RoboDK station: kr30 cnc template half inch flat end mill - paulina 3.rdk

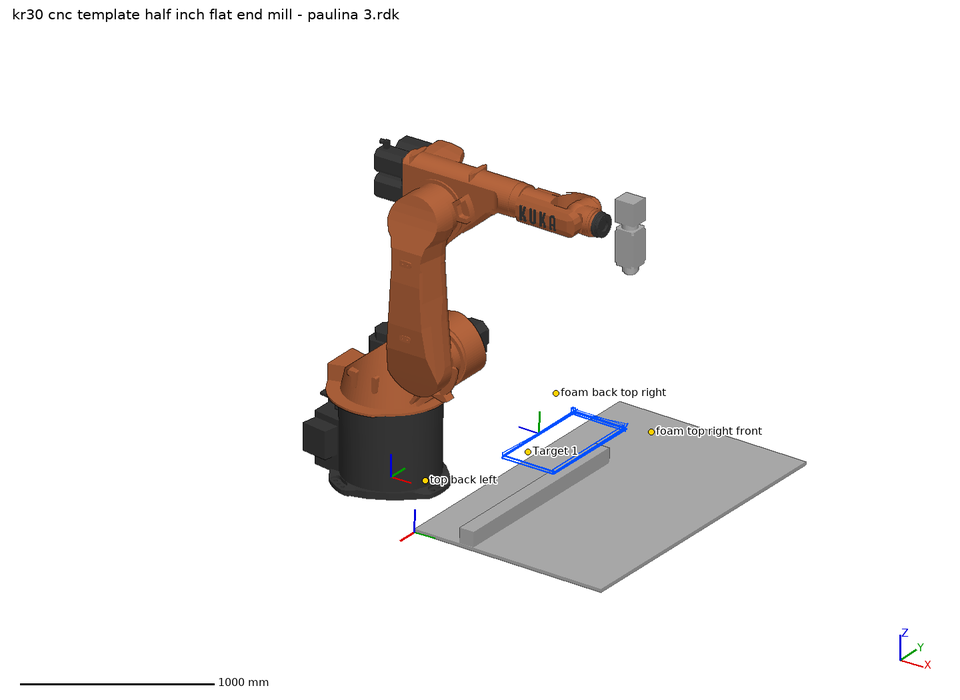
[picture v0: the station drawn from its stored meshes, robots at their saved joint values, targets as dots, program paths as lines]
Station kr30 cnc template half inch flat end mill - paulina 3. Poses are relative to the parent item; angles as X-Y-Z fixed-axis rotations.
  - frame KUKA KR 30 HA Base at (0, 0, 0) mm
    - robot KUKA KR 30 HA: 6 axes, payload 30 kg, reach 2033 mm, repeatability 0.05 mm, weight 665 kg
        modified DH rows (alpha deg, a mm, theta deg, d mm): 0, 0, 0, 815; -90, 350, 0, 0; 0, 850, -90, 0; -90, 145, 0, 820; 90, 0, 0, 0; -90, 0, 180, 170
        joint limits [-185, -135, -120, -350, -119, -350] to [185, 35, 158, 350, 119, 350]; home [0, -90, 90, 0, 0, 0]; saved at [0, -90, 90, 0, 0, 0]
      - tool rc90 spindle mm, TCP at (337.31, -2.2, 160.57) mm, size 110 x 421.3 x 118 mm, geometry from rc90 spindle mm.stl
    - frame Tabletop at (921.82, -1104.91, 385) mm, rotated rx -0.93 ry -0.21 rz -89.9 deg
      - object tabletop CHECK HEIGHT at (-1839.9, 0, 0) mm, size 1839.9 x 1168.4 x 19 mm, geometry from kr30 tabletop mm.stl
      - object kr30 pipe jig base at (-1220, -610.6, 0) mm, size 1217.6 x 88.9 x 88.9 mm, geometry from kr30 pipe jig base.stl
      - frame Frame 3 at (-550, 390, 460) mm, rotated rx 90 ry 0 rz 0 deg
        - target Target 1 (Cartesian target) at (324.46, 69.12, -153.95) mm, rotated rx -179.9 ry 0.14 rz -89.96 deg; joints [37.245, -66.694, 101.534, 53.768, -48.608, -41.204] of KUKA KR 30 HA
    - target foam back top right (Cartesian target) at (1197.65, -230.62, 906.79) mm, rotated rx -15.53 ry 90 rz -15.53 deg; joints [14.757, -102.447, 141.256, 22.791, -41.102, -17.568] of KUKA KR 30 HA
    - target foam top right front (Cartesian target) at (1797.45, -230.62, 850.68) mm, rotated rx -15.58 ry 90 rz -15.58 deg; joints [8.85, -62.405, 99.608, 14.434, -38.093, -11.451] of KUKA KR 30 HA
    - target top back left (Cartesian target) at (1223.08, -1440.01, 894.96) mm, rotated rx 58.97 ry 90 rz 58.97 deg; joints [58.171, -50.232, 76.73, 74.515, -61.834, -59.599] of KUKA KR 30 HA
  - machining project Machining Settings: C:/Users/Research Office/Downloads/b4.apt | rotZ(0) | rotX(0)*rotY(0) | roty(-90) | onStart | onPathStart | onApproach | onPoint | onRetract | onFinish | SetTool(%1) | onPathFinish
  - program Machining (938 instructions, listed below)
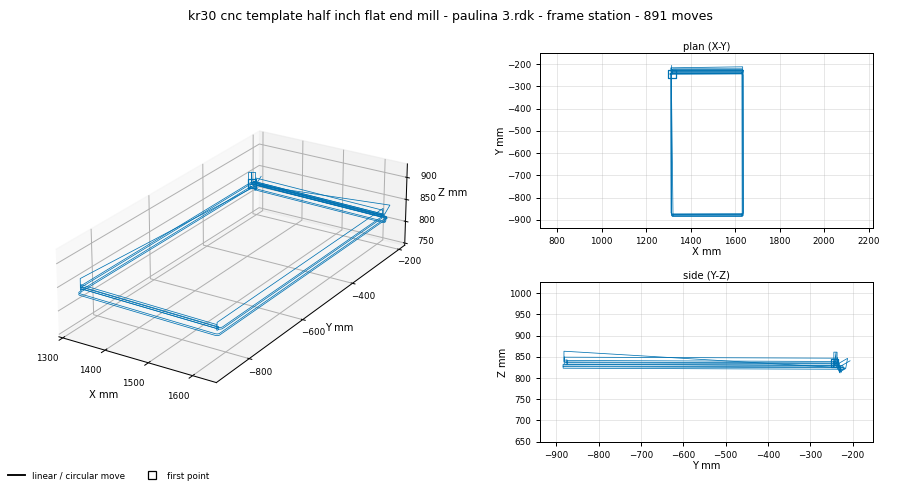
[picture p0: tool path of kr30 cnc template half inch flat end mill - paulina 3.rdk in frame station, 891 of 891 moves have a stored position in this frame; points joined in program order, loops and branches not executed]

--- program Machining (robot KUKA KR 30 HA) ---
  Smooth(10)
  Print: /'1001'
  Print: /''
  Print: /'Contour3'
  Call SetTool(1)
  Set speed (200.0 mm/s)
  Set Ref.: Frame 3
  Set Tool: rc90 spindle mm
  Show rc90 spindle mm
  MoveJ 1 to (-309.78, 0.83, 2.88) mm, rotated rx -179.88 ry 0.12 rz -89.97 deg; joints [13.585, -90.541, 136.338, 18.844, -46.545, -12.771]
  MoveL 2 to (-313.47, 25.53, 7.11) mm, rotated rx -179.9 ry 0 rz -90 deg; joints [13.435, -92.009, 135.635, -160.591, 44.341, 166.292]
  MoveL 3 to (-313.47, 25.53, 7.11) mm, rotated rx -179.9 ry 0 rz -90 deg; joints [13.435, -92.009, 135.635, -160.591, 44.341, 166.292]
  Set speed (200.0 mm/s)
  MoveL 4 to (-313.47, 10.99, 7.11) mm, rotated rx -179.9 ry 0 rz -90 deg; joints [13.441, -91.344, 136.203, -160.99, 45.507, 166.861]
  Set speed (50.0 mm/s)
  MoveL 5 to (-313.47, 4.79, 7.11) mm, rotated rx -179.9 ry 0 rz -90 deg; joints [13.444, -91.052, 136.44, -161.153, 46.008, 167.098]
  MoveL 6 to (-312.33, 3.53, 6.55) mm, rotated rx -179.9 ry 0 rz -90 deg; joints [13.5, -90.937, 136.434, -161.112, 46.125, 167.095]
  Set speed (100.0 mm/s)
  MoveL 7 to (-308.58, 3.52, 4.75) mm, rotated rx -179.9 ry 0 rz -90 deg; joints [13.681, -90.756, 136.258, -160.868, 46.171, 166.931]
  MoveC 8 to (-307.9, 3.53, 3.89) mm, rotated rx -179.9 ry 0 rz -90 deg; joints [13.707, -90.688, 136.192, -160.834, 46.179, 166.908] to (-308.14, 3.52, 2.82) mm, rotated rx -179.9 ry 0 rz -90 deg; joints [13.68, -90.62, 136.127, -160.872, 46.175, 166.934]
  MoveL 9 to (-308.14, 3.52, 2.82) mm, rotated rx -179.9 ry 0 rz -90 deg; joints [13.68, -90.62, 136.127, -160.872, 46.175, 166.934]
  MoveL 10 to (-308.36, 3.52, 2.5) mm, rotated rx -179.9 ry 0 rz -90 deg; joints [13.663, -90.603, 136.11, -160.894, 46.171, 166.95]
  MoveL 11 to (-308.56, 3.53, 2.18) mm, rotated rx -179.9 ry 0 rz -90 deg; joints [13.648, -90.584, 136.093, -160.915, 46.169, 166.964]
  MoveL 12 to (-308.73, 3.52, 1.86) mm, rotated rx -179.9 ry 0 rz -90 deg; joints [13.635, -90.566, 136.075, -160.934, 46.166, 166.977]
  MoveL 13 to (-308.88, 3.53, 1.54) mm, rotated rx -179.9 ry 0 rz -90 deg; joints [13.622, -90.547, 136.057, -160.951, 46.164, 166.989]
  MoveL 14 to (-309.02, 3.52, 1.19) mm, rotated rx -179.9 ry 0 rz -90 deg; joints [13.61, -90.526, 136.036, -160.967, 46.162, 167]
  MoveL 15 to (-309.14, 3.53, 0.84) mm, rotated rx -179.9 ry 0 rz -90 deg; joints [13.599, -90.505, 136.016, -160.983, 46.16, 167.011]
  MoveL 16 to (-309.23, 3.53, 0.5) mm, rotated rx -179.9 ry 0 rz -90 deg; joints [13.589, -90.483, 135.995, -160.996, 46.159, 167.02]
  MoveL 17 to (-309.31, 3.53, 0.15) mm, rotated rx -179.9 ry 0 rz -90 deg; joints [13.58, -90.461, 135.973, -161.008, 46.157, 167.029]
  MoveL 18 to (-309.36, 3.53, -0.2) mm, rotated rx -179.9 ry 0 rz -90 deg; joints [13.573, -90.438, 135.952, -161.018, 46.156, 167.036]
  MoveL 19 to (-309.4, 3.52, -0.55) mm, rotated rx -179.9 ry 0 rz -90 deg; joints [13.566, -90.416, 135.93, -161.027, 46.156, 167.042]
  MoveL 20 to (-309.41, 3.53, -1.25) mm, rotated rx -179.9 ry 0 rz -90 deg; joints [13.556, -90.369, 135.885, -161.041, 46.155, 167.052]
  MoveL 21 to (-309.41, 3.52, -310.99) mm, rotated rx -179.9 ry 0 rz -90 deg; joints [10.396, -71.401, 113.657, -164.475, 42.367, 168.785]
  MoveL 22 to (-309.4, 3.52, -311.68) mm, rotated rx -179.9 ry 0 rz -90 deg; joints [10.391, -71.36, 113.601, -164.478, 42.352, 168.784]
  MoveL 23 to (-309.36, 3.52, -312.03) mm, rotated rx -179.9 ry 0 rz -90 deg; joints [10.39, -71.34, 113.573, -164.478, 42.344, 168.783]
  MoveL 24 to (-309.31, 3.52, -312.38) mm, rotated rx -179.9 ry 0 rz -90 deg; joints [10.389, -71.319, 113.545, -164.476, 42.337, 168.78]
  MoveL 25 to (-309.23, 3.53, -312.73) mm, rotated rx -179.9 ry 0 rz -90 deg; joints [10.39, -71.298, 113.516, -164.473, 42.329, 168.777]
  MoveL 26 to (-309.14, 3.52, -313.08) mm, rotated rx -179.9 ry 0 rz -90 deg; joints [10.391, -71.276, 113.487, -164.469, 42.322, 168.772]
  MoveL 27 to (-309.02, 3.52, -313.43) mm, rotated rx -179.9 ry 0 rz -90 deg; joints [10.393, -71.255, 113.457, -164.464, 42.315, 168.767]
  MoveL 28 to (-308.88, 3.52, -313.78) mm, rotated rx -179.9 ry 0 rz -90 deg; joints [10.396, -71.233, 113.427, -164.457, 42.308, 168.76]
  MoveL 29 to (-308.73, 3.53, -314.1) mm, rotated rx -179.9 ry 0 rz -90 deg; joints [10.4, -71.213, 113.4, -164.449, 42.301, 168.753]
  MoveL 30 to (-308.56, 3.52, -314.42) mm, rotated rx -179.9 ry 0 rz -90 deg; joints [10.405, -71.192, 113.372, -164.439, 42.295, 168.745]
  MoveL 31 to (-308.36, 3.52, -314.73) mm, rotated rx -179.9 ry 0 rz -90 deg; joints [10.411, -71.172, 113.343, -164.429, 42.289, 168.736]
  MoveL 32 to (-308.14, 3.52, -315.05) mm, rotated rx -179.9 ry 0 rz -90 deg; joints [10.418, -71.151, 113.315, -164.416, 42.283, 168.725]
  MoveL 33 to (-307.96, 3.52, -315.28) mm, rotated rx -179.9 ry 0 rz -90 deg; joints [10.424, -71.136, 113.294, -164.406, 42.278, 168.717]
  MoveL 34 to (-307.77, 3.53, -315.5) mm, rotated rx -179.9 ry 0 rz -90 deg; joints [10.43, -71.121, 113.274, -164.395, 42.274, 168.708]
  MoveL 35 to (-307.55, 3.53, -315.73) mm, rotated rx -179.9 ry 0 rz -90 deg; joints [10.438, -71.105, 113.252, -164.382, 42.27, 168.697]
  MoveL 36 to (-307.32, 3.53, -315.94) mm, rotated rx -179.9 ry 0 rz -90 deg; joints [10.445, -71.09, 113.232, -164.369, 42.266, 168.687]
  MoveL 37 to (-306.92, 3.52, -316.28) mm, rotated rx -179.9 ry 0 rz -90 deg; joints [10.46, -71.066, 113.198, -164.346, 42.26, 168.668]
  MoveL 38 to (-306.51, 3.53, -316.57) mm, rotated rx -179.9 ry 0 rz -90 deg; joints [10.475, -71.045, 113.17, -164.321, 42.256, 168.649]
  MoveL 39 to (-306.22, 3.52, -316.74) mm, rotated rx -179.9 ry 0 rz -90 deg; joints [10.486, -71.032, 113.151, -164.304, 42.253, 168.635]
  MoveL 40 to (-305.93, 3.52, -316.9) mm, rotated rx -179.9 ry 0 rz -90 deg; joints [10.497, -71.02, 113.134, -164.287, 42.251, 168.621]
  MoveL 41 to (-305.64, 3.52, -317.04) mm, rotated rx -179.9 ry 0 rz -90 deg; joints [10.508, -71.009, 113.119, -164.269, 42.249, 168.608]
  MoveL 42 to (-305.35, 3.52, -317.16) mm, rotated rx -179.9 ry 0 rz -90 deg; joints [10.519, -70.999, 113.105, -164.251, 42.248, 168.594]
  MoveL 43 to (-305, 3.52, -317.28) mm, rotated rx -179.9 ry 0 rz -90 deg; joints [10.533, -70.988, 113.09, -164.23, 42.246, 168.578]
  MoveL 44 to (-304.65, 3.52, -317.38) mm, rotated rx -179.9 ry 0 rz -90 deg; joints [10.547, -70.978, 113.076, -164.209, 42.245, 168.562]
  MoveL 45 to (-304.3, 3.52, -317.46) mm, rotated rx -179.9 ry 0 rz -90 deg; joints [10.561, -70.97, 113.065, -164.187, 42.245, 168.545]
  MoveL 46 to (-303.95, 3.53, -317.52) mm, rotated rx -179.9 ry 0 rz -90 deg; joints [10.575, -70.963, 113.055, -164.166, 42.245, 168.529]
  MoveL 47 to (-303.6, 3.52, -317.56) mm, rotated rx -179.9 ry 0 rz -90 deg; joints [10.59, -70.956, 113.046, -164.144, 42.246, 168.513]
  MoveL 48 to (-303.26, 3.52, -317.58) mm, rotated rx -179.9 ry 0 rz -90 deg; joints [10.604, -70.952, 113.039, -164.122, 42.247, 168.496]
  MoveL 49 to (-302.56, 3.53, -317.59) mm, rotated rx -179.9 ry 0 rz -90 deg; joints [10.634, -70.944, 113.028, -164.078, 42.25, 168.464]
  MoveL 50 to (315.11, 3.52, -317.59) mm, rotated rx -179.9 ry 0 rz -90 deg; joints [33.369, -56.917, 91.684, -130.086, 45.952, 141.267]
  MoveL 51 to (315.8, 3.53, -317.58) mm, rotated rx -179.9 ry 0 rz -90 deg; joints [33.39, -56.894, 91.646, -130.052, 45.956, 141.236]
  MoveL 52 to (316.15, 3.53, -317.56) mm, rotated rx -179.9 ry 0 rz -90 deg; joints [33.401, -56.883, 91.628, -130.035, 45.958, 141.221]
  MoveL 53 to (316.5, 3.52, -317.52) mm, rotated rx -179.9 ry 0 rz -90 deg; joints [33.413, -56.873, 91.612, -130.018, 45.961, 141.206]
  MoveL 54 to (316.82, 3.52, -317.46) mm, rotated rx -179.9 ry 0 rz -90 deg; joints [33.423, -56.865, 91.599, -130.003, 45.965, 141.192]
  MoveL 55 to (317.13, 3.52, -317.39) mm, rotated rx -179.9 ry 0 rz -90 deg; joints [33.434, -56.858, 91.588, -129.988, 45.969, 141.18]
  MoveL 56 to (317.45, 3.53, -317.3) mm, rotated rx -179.9 ry 0 rz -90 deg; joints [33.446, -56.852, 91.578, -129.973, 45.974, 141.167]
  MoveL 57 to (317.76, 3.52, -317.2) mm, rotated rx -179.9 ry 0 rz -90 deg; joints [33.457, -56.847, 91.569, -129.957, 45.979, 141.155]
  MoveL 58 to (318.08, 3.52, -317.07) mm, rotated rx -179.9 ry 0 rz -90 deg; joints [33.469, -56.843, 91.562, -129.942, 45.985, 141.143]
  MoveL 59 to (318.4, 3.52, -316.93) mm, rotated rx -179.9 ry 0 rz -90 deg; joints [33.482, -56.839, 91.557, -129.927, 45.991, 141.131]
  MoveL 60 to (318.71, 3.52, -316.76) mm, rotated rx -179.9 ry 0 rz -90 deg; joints [33.495, -56.837, 91.553, -129.912, 45.998, 141.12]
  MoveL 61 to (319.03, 3.53, -316.57) mm, rotated rx -179.9 ry 0 rz -90 deg; joints [33.508, -56.836, 91.551, -129.897, 46.006, 141.109]
  MoveL 62 to (319.29, 3.52, -316.39) mm, rotated rx -179.9 ry 0 rz -90 deg; joints [33.52, -56.837, 91.552, -129.884, 46.013, 141.101]
  MoveL 63 to (319.63, 3.52, -316.13) mm, rotated rx -179.9 ry 0 rz -90 deg; joints [33.535, -56.839, 91.554, -129.868, 46.024, 141.09]
  MoveL 64 to (319.96, 3.52, -315.83) mm, rotated rx -179.9 ry 0 rz -90 deg; joints [33.552, -56.843, 91.56, -129.852, 46.035, 141.081]
  MoveL 65 to (320.32, 3.53, -315.46) mm, rotated rx -179.9 ry 0 rz -90 deg; joints [33.57, -56.85, 91.571, -129.835, 46.049, 141.071]
  MoveL 66 to (320.63, 3.52, -315.08) mm, rotated rx -179.9 ry 0 rz -90 deg; joints [33.587, -56.859, 91.585, -129.82, 46.063, 141.064]
  MoveL 67 to (320.86, 3.52, -314.76) mm, rotated rx -179.9 ry 0 rz -90 deg; joints [33.601, -56.868, 91.599, -129.809, 46.075, 141.059]
  MoveL 68 to (321.07, 3.52, -314.43) mm, rotated rx -179.9 ry 0 rz -90 deg; joints [33.614, -56.878, 91.615, -129.8, 46.087, 141.056]
  MoveL 69 to (321.24, 3.53, -314.1) mm, rotated rx -179.9 ry 0 rz -90 deg; joints [33.626, -56.889, 91.632, -129.792, 46.098, 141.054]
  MoveL 70 to (321.4, 3.52, -313.78) mm, rotated rx -179.9 ry 0 rz -90 deg; joints [33.637, -56.9, 91.65, -129.784, 46.11, 141.053]
  MoveL 71 to (321.54, 3.52, -313.43) mm, rotated rx -179.9 ry 0 rz -90 deg; joints [33.648, -56.914, 91.671, -129.778, 46.122, 141.053]
  MoveL 72 to (321.66, 3.52, -313.08) mm, rotated rx -179.9 ry 0 rz -90 deg; joints [33.659, -56.928, 91.694, -129.773, 46.134, 141.054]
  MoveL 73 to (321.75, 3.52, -312.73) mm, rotated rx -179.9 ry 0 rz -90 deg; joints [33.669, -56.943, 91.717, -129.768, 46.145, 141.056]
  MoveL 74 to (321.83, 3.52, -312.38) mm, rotated rx -179.9 ry 0 rz -90 deg; joints [33.678, -56.958, 91.742, -129.765, 46.157, 141.059]
  MoveL 75 to (321.88, 3.52, -312.03) mm, rotated rx -179.9 ry 0 rz -90 deg; joints [33.687, -56.974, 91.767, -129.763, 46.169, 141.062]
  MoveL 76 to (321.91, 3.52, -311.68) mm, rotated rx -179.9 ry 0 rz -90 deg; joints [33.695, -56.991, 91.794, -129.761, 46.18, 141.067]
  MoveL 77 to (321.93, 3.53, -310.99) mm, rotated rx -179.9 ry 0 rz -90 deg; joints [33.71, -57.027, 91.851, -129.761, 46.203, 141.079]
  MoveL 78 to (321.93, 3.52, -1.25) mm, rotated rx -179.9 ry 0 rz -90 deg; joints [41.195, -71.851, 113.68, -126.635, 55.146, 143.485]
  MoveL 79 to (321.91, 3.52, -0.55) mm, rotated rx -179.9 ry 0 rz -90 deg; joints [41.215, -71.883, 113.723, -126.623, 55.164, 143.485]
  MoveL 80 to (321.88, 3.52, -0.2) mm, rotated rx -179.9 ry 0 rz -90 deg; joints [41.224, -71.9, 113.746, -126.617, 55.173, 143.486]
  MoveL 81 to (321.83, 3.52, 0.15) mm, rotated rx -179.9 ry 0 rz -90 deg; joints [41.232, -71.918, 113.77, -126.613, 55.181, 143.488]
  MoveL 82 to (321.75, 3.52, 0.5) mm, rotated rx -179.9 ry 0 rz -90 deg; joints [41.239, -71.936, 113.795, -126.609, 55.19, 143.49]
  MoveL 83 to (321.66, 3.53, 0.84) mm, rotated rx -179.9 ry 0 rz -90 deg; joints [41.246, -71.956, 113.821, -126.606, 55.198, 143.493]
  MoveL 84 to (321.54, 3.53, 1.19) mm, rotated rx -179.9 ry 0 rz -90 deg; joints [41.252, -71.976, 113.848, -126.604, 55.206, 143.496]
  MoveL 85 to (321.4, 3.53, 1.54) mm, rotated rx -179.9 ry 0 rz -90 deg; joints [41.258, -71.997, 113.877, -126.603, 55.213, 143.501]
  MoveL 86 to (321.24, 3.52, 1.87) mm, rotated rx -179.9 ry 0 rz -90 deg; joints [41.262, -72.017, 113.904, -126.602, 55.22, 143.505]
  MoveL 87 to (321.07, 3.52, 2.19) mm, rotated rx -179.9 ry 0 rz -90 deg; joints [41.266, -72.039, 113.934, -126.603, 55.227, 143.511]
  MoveL 88 to (320.86, 3.52, 2.52) mm, rotated rx -179.9 ry 0 rz -90 deg; joints [41.269, -72.061, 113.964, -126.605, 55.233, 143.517]
  MoveL 89 to (320.63, 3.52, 2.85) mm, rotated rx -179.9 ry 0 rz -90 deg; joints [41.27, -72.085, 113.996, -126.608, 55.239, 143.524]
  MoveL 90 to (320.32, 3.52, 3.22) mm, rotated rx -179.9 ry 0 rz -90 deg; joints [41.271, -72.114, 114.035, -126.613, 55.246, 143.534]
  MoveL 91 to (319.96, 3.52, 3.6) mm, rotated rx -179.9 ry 0 rz -90 deg; joints [41.27, -72.145, 114.077, -126.62, 55.252, 143.545]
  MoveL 92 to (319.63, 3.53, 3.89) mm, rotated rx -179.9 ry 0 rz -90 deg; joints [41.268, -72.171, 114.113, -126.628, 55.256, 143.556]
  MoveL 93 to (319.29, 3.52, 4.15) mm, rotated rx -179.9 ry 0 rz -90 deg; joints [41.264, -72.196, 114.146, -126.636, 55.259, 143.566]
  MoveL 94 to (319.03, 3.53, 4.33) mm, rotated rx -179.9 ry 0 rz -90 deg; joints [41.261, -72.214, 114.171, -126.643, 55.261, 143.575]
  MoveL 95 to (318.71, 3.52, 4.52) mm, rotated rx -179.9 ry 0 rz -90 deg; joints [41.256, -72.235, 114.2, -126.652, 55.263, 143.585]
  MoveL 96 to (318.4, 3.52, 4.69) mm, rotated rx -179.9 ry 0 rz -90 deg; joints [41.25, -72.255, 114.226, -126.661, 55.264, 143.594]
  MoveL 97 to (318.08, 3.53, 4.84) mm, rotated rx -179.9 ry 0 rz -90 deg; joints [41.244, -72.274, 114.252, -126.671, 55.264, 143.604]
  MoveL 98 to (317.76, 3.53, 4.96) mm, rotated rx -179.9 ry 0 rz -90 deg; joints [41.237, -72.291, 114.276, -126.681, 55.264, 143.614]
  MoveL 99 to (317.45, 3.52, 5.07) mm, rotated rx -179.9 ry 0 rz -90 deg; joints [41.23, -72.308, 114.3, -126.692, 55.263, 143.624]
  MoveL 100 to (317.13, 3.53, 5.16) mm, rotated rx -179.9 ry 0 rz -90 deg; joints [41.222, -72.325, 114.322, -126.703, 55.262, 143.634]
  MoveL 101 to (316.82, 3.52, 5.23) mm, rotated rx -179.9 ry 0 rz -90 deg; joints [41.214, -72.34, 114.343, -126.714, 55.261, 143.644]
  MoveL 102 to (316.5, 3.52, 5.28) mm, rotated rx -179.9 ry 0 rz -90 deg; joints [41.205, -72.355, 114.363, -126.725, 55.259, 143.654]
  MoveL 103 to (316.15, 3.53, 5.32) mm, rotated rx -179.9 ry 0 rz -90 deg; joints [41.195, -72.37, 114.384, -126.739, 55.256, 143.665]
  MoveL 104 to (315.8, 3.53, 5.35) mm, rotated rx -179.9 ry 0 rz -90 deg; joints [41.184, -72.385, 114.404, -126.752, 55.253, 143.676]
  MoveL 105 to (315.11, 3.53, 5.35) mm, rotated rx -179.9 ry 0 rz -90 deg; joints [41.162, -72.412, 114.441, -126.78, 55.245, 143.699]
  MoveL 106 to (-302.56, 3.53, 5.35) mm, rotated rx -179.9 ry 0 rz -90 deg; joints [14.019, -90.699, 136.199, -160.413, 46.247, 166.621]
  MoveL 107 to (-303.26, 3.53, 5.35) mm, rotated rx -179.9 ry 0 rz -90 deg; joints [13.981, -90.71, 136.21, -160.465, 46.238, 166.656]
  MoveL 108 to (-303.6, 3.52, 5.33) mm, rotated rx -179.9 ry 0 rz -90 deg; joints [13.961, -90.714, 136.215, -160.491, 46.234, 166.674]
  MoveL 109 to (-303.95, 3.52, 5.29) mm, rotated rx -179.9 ry 0 rz -90 deg; joints [13.942, -90.717, 136.218, -160.517, 46.229, 166.692]
  MoveL 110 to (-304.3, 3.53, 5.23) mm, rotated rx -179.9 ry 0 rz -90 deg; joints [13.922, -90.719, 136.22, -160.544, 46.225, 166.71]
  MoveL 111 to (-304.65, 3.53, 5.15) mm, rotated rx -179.9 ry 0 rz -90 deg; joints [13.902, -90.72, 136.221, -160.571, 46.22, 166.728]
  MoveL 112 to (-305, 3.53, 5.05) mm, rotated rx -179.9 ry 0 rz -90 deg; joints [13.881, -90.718, 136.22, -160.599, 46.216, 166.747]
  MoveL 113 to (-305.35, 3.52, 4.92) mm, rotated rx -179.9 ry 0 rz -90 deg; joints [13.861, -90.716, 136.217, -160.627, 46.211, 166.766]
  MoveL 114 to (-305.64, 3.53, 4.8) mm, rotated rx -179.9 ry 0 rz -90 deg; joints [13.843, -90.713, 136.214, -160.65, 46.208, 166.783]
  MoveL 115 to (-305.93, 3.53, 4.67) mm, rotated rx -179.9 ry 0 rz -90 deg; joints [13.825, -90.708, 136.21, -160.674, 46.204, 166.799]
  MoveL 116 to (-306.22, 3.52, 4.51) mm, rotated rx -179.9 ry 0 rz -90 deg; joints [13.807, -90.702, 136.205, -160.699, 46.2, 166.816]
  MoveL 117 to (-306.51, 3.52, 4.33) mm, rotated rx -179.9 ry 0 rz -90 deg; joints [13.789, -90.695, 136.198, -160.723, 46.196, 166.833]
  MoveL 118 to (-306.92, 3.53, 4.05) mm, rotated rx -179.9 ry 0 rz -90 deg; joints [13.763, -90.683, 136.186, -160.759, 46.191, 166.857]
  MoveL 119 to (-307.32, 3.53, 3.71) mm, rotated rx -179.9 ry 0 rz -90 deg; joints [13.736, -90.667, 136.171, -160.795, 46.186, 166.882]
  MoveL 120 to (-307.55, 3.52, 3.5) mm, rotated rx -179.9 ry 0 rz -90 deg; joints [13.721, -90.656, 136.161, -160.816, 46.183, 166.896]
  MoveL 121 to (-307.77, 3.52, 3.26) mm, rotated rx -179.9 ry 0 rz -90 deg; joints [13.706, -90.644, 136.15, -160.836, 46.18, 166.91]
  MoveL 122 to (-307.96, 3.53, 3.04) mm, rotated rx -179.9 ry 0 rz -90 deg; joints [13.692, -90.632, 136.138, -160.855, 46.177, 166.923]
  MoveL 123 to (-308.14, 3.52, 2.82) mm, rotated rx -179.9 ry 0 rz -90 deg; joints [13.68, -90.62, 136.127, -160.872, 46.175, 166.934]
  MoveC 124 to (-309.89, 3.53, 2.59) mm, rotated rx -179.9 ry 0 rz -90 deg; joints [13.581, -90.633, 136.14, -161.006, 46.153, 167.026] to (-310.17, 3.53, 4.33) mm, rotated rx -179.9 ry 0 rz -90 deg; joints [13.589, -90.754, 136.257, -160.994, 46.15, 167.017]
  MoveL 125 to (-310.17, 3.52, 4.33) mm, rotated rx -179.9 ry 0 rz -90 deg; joints [13.589, -90.754, 136.257, -160.994, 46.15, 167.017]
  MoveL 126 to (-309.48, 3.53, 5.32) mm, rotated rx -179.9 ry 0 rz -90 deg; joints [13.64, -90.809, 136.31, -160.924, 46.16, 166.968]
  Set speed (50.0 mm/s)
  MoveL 127 to (-309.48, 1.27, 5.32) mm, rotated rx -179.9 ry 0 rz -90 deg; joints [13.641, -90.701, 136.395, -160.983, 46.342, 167.055]
  MoveL 128 to (-308.44, 0, 4.59) mm, rotated rx -179.9 ry 0 rz -90 deg; joints [13.688, -90.575, 136.379, -160.953, 46.457, 167.061]
  Set speed (100.0 mm/s)
  MoveC 129 to (-307.92, 0, 3.77) mm, rotated rx -179.9 ry 0 rz -90 deg; joints [13.706, -90.512, 136.317, -160.93, 46.462, 167.046] to (-308.14, 0, 2.82) mm, rotated rx -179.9 ry 0 rz -90 deg; joints [13.681, -90.452, 136.259, -160.964, 46.459, 167.069]
  MoveL 130 to (-308.14, 0, 2.82) mm, rotated rx -179.9 ry 0 rz -90 deg; joints [13.681, -90.452, 136.259, -160.964, 46.459, 167.069]
  MoveL 131 to (-308.36, 0, 2.5) mm, rotated rx -179.9 ry 0 rz -90 deg; joints [13.665, -90.435, 136.242, -160.986, 46.456, 167.084]
  MoveL 132 to (-308.56, 0, 2.18) mm, rotated rx -179.9 ry 0 rz -90 deg; joints [13.65, -90.417, 136.225, -161.007, 46.453, 167.098]
  MoveL 133 to (-308.73, 0, 1.86) mm, rotated rx -179.9 ry 0 rz -90 deg; joints [13.636, -90.398, 136.207, -161.025, 46.45, 167.111]
  MoveL 134 to (-308.88, 0, 1.54) mm, rotated rx -179.9 ry 0 rz -90 deg; joints [13.624, -90.379, 136.189, -161.042, 46.448, 167.123]
  MoveL 135 to (-309.02, 0, 1.19) mm, rotated rx -179.9 ry 0 rz -90 deg; joints [13.611, -90.358, 136.169, -161.059, 46.446, 167.134]
  MoveL 136 to (-309.14, 0, 0.84) mm, rotated rx -179.9 ry 0 rz -90 deg; joints [13.6, -90.337, 136.148, -161.074, 46.444, 167.144]
  MoveL 137 to (-309.23, 0, 0.5) mm, rotated rx -179.9 ry 0 rz -90 deg; joints [13.591, -90.315, 136.127, -161.087, 46.443, 167.154]
  MoveL 138 to (-309.31, 0, 0.15) mm, rotated rx -179.9 ry 0 rz -90 deg; joints [13.582, -90.293, 136.106, -161.099, 46.441, 167.162]
  MoveL 139 to (-309.36, 0, -0.2) mm, rotated rx -179.9 ry 0 rz -90 deg; joints [13.574, -90.271, 136.084, -161.109, 46.44, 167.169]
  MoveL 140 to (-309.4, 0, -0.55) mm, rotated rx -179.9 ry 0 rz -90 deg; joints [13.568, -90.248, 136.062, -161.118, 46.439, 167.175]
  MoveL 141 to (-309.41, 0, -1.25) mm, rotated rx -179.9 ry 0 rz -90 deg; joints [13.558, -90.202, 136.017, -161.132, 46.438, 167.185]
  MoveL 142 to (-309.41, 0, -310.99) mm, rotated rx -179.9 ry 0 rz -90 deg; joints [10.397, -71.274, 113.767, -164.543, 42.596, 168.878]
  MoveL 143 to (-309.4, 0, -311.68) mm, rotated rx -179.9 ry 0 rz -90 deg; joints [10.392, -71.233, 113.711, -164.546, 42.581, 168.877]
  MoveL 144 to (-309.36, 0, -312.03) mm, rotated rx -179.9 ry 0 rz -90 deg; joints [10.391, -71.212, 113.683, -164.546, 42.573, 168.876]
  MoveL 145 to (-309.31, 0, -312.38) mm, rotated rx -179.9 ry 0 rz -90 deg; joints [10.39, -71.191, 113.655, -164.544, 42.566, 168.873]
  MoveL 146 to (-309.23, 0, -312.73) mm, rotated rx -179.9 ry 0 rz -90 deg; joints [10.391, -71.17, 113.626, -164.541, 42.558, 168.869]
  MoveL 147 to (-309.14, 0, -313.08) mm, rotated rx -179.9 ry 0 rz -90 deg; joints [10.392, -71.149, 113.597, -164.537, 42.551, 168.865]
  MoveL 148 to (-309.02, 0, -313.43) mm, rotated rx -179.9 ry 0 rz -90 deg; joints [10.394, -71.127, 113.567, -164.531, 42.544, 168.86]
  MoveL 149 to (-308.88, 0, -313.78) mm, rotated rx -179.9 ry 0 rz -90 deg; joints [10.397, -71.106, 113.537, -164.524, 42.537, 168.853]
  MoveL 150 to (-308.73, 0, -314.1) mm, rotated rx -179.9 ry 0 rz -90 deg; joints [10.401, -71.086, 113.51, -164.517, 42.53, 168.846]
  MoveL 151 to (-308.56, 0, -314.42) mm, rotated rx -179.9 ry 0 rz -90 deg; joints [10.406, -71.065, 113.482, -164.508, 42.524, 168.838]
  MoveL 152 to (-308.36, 0, -314.73) mm, rotated rx -179.9 ry 0 rz -90 deg; joints [10.412, -71.045, 113.453, -164.497, 42.517, 168.829]
  MoveL 153 to (-308.14, 0, -315.05) mm, rotated rx -179.9 ry 0 rz -90 deg; joints [10.419, -71.024, 113.425, -164.484, 42.511, 168.818]
  MoveL 154 to (-307.96, 0, -315.28) mm, rotated rx -179.9 ry 0 rz -90 deg; joints [10.425, -71.009, 113.404, -164.474, 42.507, 168.81]
  MoveL 155 to (-307.77, 0, -315.5) mm, rotated rx -179.9 ry 0 rz -90 deg; joints [10.431, -70.994, 113.384, -164.463, 42.503, 168.801]
  MoveL 156 to (-307.55, 0, -315.73) mm, rotated rx -179.9 ry 0 rz -90 deg; joints [10.439, -70.978, 113.362, -164.451, 42.498, 168.791]
  MoveL 157 to (-307.32, 0, -315.94) mm, rotated rx -179.9 ry 0 rz -90 deg; joints [10.446, -70.963, 113.341, -164.438, 42.495, 168.78]
  MoveL 158 to (-306.92, 0, -316.28) mm, rotated rx -179.9 ry 0 rz -90 deg; joints [10.461, -70.939, 113.308, -164.414, 42.489, 168.761]
  MoveL 159 to (-306.51, 0, -316.57) mm, rotated rx -179.9 ry 0 rz -90 deg; joints [10.476, -70.918, 113.279, -164.39, 42.484, 168.742]
  MoveL 160 to (-306.22, 0, -316.74) mm, rotated rx -179.9 ry 0 rz -90 deg; joints [10.487, -70.905, 113.261, -164.373, 42.481, 168.729]
  MoveL 161 to (-305.93, 0, -316.9) mm, rotated rx -179.9 ry 0 rz -90 deg; joints [10.498, -70.893, 113.244, -164.355, 42.479, 168.715]
  MoveL 162 to (-305.64, 0, -317.04) mm, rotated rx -179.9 ry 0 rz -90 deg; joints [10.509, -70.882, 113.229, -164.338, 42.477, 168.702]
  MoveL 163 to (-305.35, 0, -317.16) mm, rotated rx -179.9 ry 0 rz -90 deg; joints [10.52, -70.872, 113.215, -164.32, 42.475, 168.688]
  MoveL 164 to (-305, 0, -317.28) mm, rotated rx -179.9 ry 0 rz -90 deg; joints [10.534, -70.861, 113.2, -164.299, 42.474, 168.672]
  MoveL 165 to (-304.65, 0, -317.38) mm, rotated rx -179.9 ry 0 rz -90 deg; joints [10.548, -70.851, 113.186, -164.278, 42.473, 168.656]
  MoveL 166 to (-304.3, 0, -317.46) mm, rotated rx -179.9 ry 0 rz -90 deg; joints [10.562, -70.843, 113.175, -164.256, 42.473, 168.64]
  MoveL 167 to (-303.95, 0, -317.52) mm, rotated rx -179.9 ry 0 rz -90 deg; joints [10.576, -70.836, 113.164, -164.235, 42.473, 168.624]
  MoveL 168 to (-303.6, 0, -317.56) mm, rotated rx -179.9 ry 0 rz -90 deg; joints [10.591, -70.83, 113.156, -164.213, 42.474, 168.607]
  MoveL 169 to (-303.26, 0, -317.58) mm, rotated rx -179.9 ry 0 rz -90 deg; joints [10.605, -70.825, 113.149, -164.191, 42.475, 168.591]
  MoveL 170 to (-302.56, 0, -317.59) mm, rotated rx -179.9 ry 0 rz -90 deg; joints [10.635, -70.817, 113.138, -164.148, 42.477, 168.559]
  MoveL 171 to (315.11, 0, -317.59) mm, rotated rx -179.9 ry 0 rz -90 deg; joints [33.37, -56.819, 91.792, -130.237, 46.086, 141.486]
  MoveL 172 to (315.8, 0, -317.58) mm, rotated rx -179.9 ry 0 rz -90 deg; joints [33.392, -56.795, 91.754, -130.203, 46.09, 141.454]
  MoveL 173 to (316.15, 0, -317.56) mm, rotated rx -179.9 ry 0 rz -90 deg; joints [33.403, -56.785, 91.737, -130.186, 46.092, 141.439]
  MoveL 174 to (316.5, 0, -317.52) mm, rotated rx -179.9 ry 0 rz -90 deg; joints [33.414, -56.775, 91.721, -130.169, 46.095, 141.424]
  MoveL 175 to (316.82, 0, -317.46) mm, rotated rx -179.9 ry 0 rz -90 deg; joints [33.425, -56.767, 91.708, -130.154, 46.099, 141.411]
  MoveL 176 to (317.13, 0, -317.39) mm, rotated rx -179.9 ry 0 rz -90 deg; joints [33.436, -56.76, 91.696, -130.139, 46.103, 141.398]
  MoveL 177 to (317.45, 0, -317.3) mm, rotated rx -179.9 ry 0 rz -90 deg; joints [33.447, -56.754, 91.686, -130.123, 46.108, 141.386]
  MoveL 178 to (317.76, 0, -317.2) mm, rotated rx -179.9 ry 0 rz -90 deg; joints [33.459, -56.749, 91.678, -130.108, 46.113, 141.373]
  MoveL 179 to (318.08, 0, -317.07) mm, rotated rx -179.9 ry 0 rz -90 deg; joints [33.471, -56.744, 91.67, -130.093, 46.118, 141.361]
  MoveL 180 to (318.4, 0, -316.93) mm, rotated rx -179.9 ry 0 rz -90 deg; joints [33.484, -56.741, 91.665, -130.078, 46.125, 141.35]
  MoveL 181 to (318.71, 0, -316.76) mm, rotated rx -179.9 ry 0 rz -90 deg; joints [33.497, -56.739, 91.661, -130.063, 46.132, 141.339]
  MoveL 182 to (319.03, 0, -316.57) mm, rotated rx -179.9 ry 0 rz -90 deg; joints [33.51, -56.738, 91.66, -130.048, 46.14, 141.328]
  MoveL 183 to (319.29, 0, -316.39) mm, rotated rx -179.9 ry 0 rz -90 deg; joints [33.522, -56.739, 91.66, -130.035, 46.147, 141.319]
  MoveL 184 to (319.63, 0, -316.13) mm, rotated rx -179.9 ry 0 rz -90 deg; joints [33.537, -56.741, 91.663, -130.019, 46.157, 141.309]
  MoveL 185 to (319.96, 0, -315.83) mm, rotated rx -179.9 ry 0 rz -90 deg; joints [33.553, -56.745, 91.669, -130.003, 46.169, 141.299]
  MoveL 186 to (320.32, 0, -315.46) mm, rotated rx -179.9 ry 0 rz -90 deg; joints [33.572, -56.752, 91.68, -129.986, 46.183, 141.29]
  MoveL 187 to (320.63, 0, -315.08) mm, rotated rx -179.9 ry 0 rz -90 deg; joints [33.589, -56.761, 91.694, -129.971, 46.197, 141.283]
  MoveL 188 to (320.86, 0, -314.76) mm, rotated rx -179.9 ry 0 rz -90 deg; joints [33.602, -56.77, 91.708, -129.96, 46.208, 141.278]
  MoveL 189 to (321.07, 0, -314.43) mm, rotated rx -179.9 ry 0 rz -90 deg; joints [33.615, -56.78, 91.723, -129.951, 46.22, 141.275]
  MoveL 190 to (321.24, 0, -314.1) mm, rotated rx -179.9 ry 0 rz -90 deg; joints [33.627, -56.79, 91.74, -129.942, 46.232, 141.273]
  MoveL 191 to (321.4, 0, -313.78) mm, rotated rx -179.9 ry 0 rz -90 deg; joints [33.638, -56.802, 91.759, -129.935, 46.243, 141.272]
  MoveL 192 to (321.54, 0, -313.43) mm, rotated rx -179.9 ry 0 rz -90 deg; joints [33.65, -56.815, 91.78, -129.929, 46.255, 141.272]
  MoveL 193 to (321.66, 0, -313.08) mm, rotated rx -179.9 ry 0 rz -90 deg; joints [33.66, -56.829, 91.802, -129.923, 46.267, 141.273]
  MoveL 194 to (321.75, 0, -312.73) mm, rotated rx -179.9 ry 0 rz -90 deg; joints [33.67, -56.844, 91.825, -129.919, 46.279, 141.275]
  MoveL 195 to (321.83, 0, -312.38) mm, rotated rx -179.9 ry 0 rz -90 deg; joints [33.68, -56.86, 91.85, -129.915, 46.291, 141.277]
  MoveL 196 to (321.88, 0, -312.03) mm, rotated rx -179.9 ry 0 rz -90 deg; joints [33.688, -56.876, 91.876, -129.913, 46.302, 141.281]
  MoveL 197 to (321.91, 0, -311.68) mm, rotated rx -179.9 ry 0 rz -90 deg; joints [33.696, -56.893, 91.903, -129.912, 46.314, 141.286]
  MoveL 198 to (321.93, 0, -310.99) mm, rotated rx -179.9 ry 0 rz -90 deg; joints [33.711, -56.928, 91.959, -129.911, 46.336, 141.297]
  MoveL 199 to (321.93, 0, -1.25) mm, rotated rx -179.9 ry 0 rz -90 deg; joints [41.197, -71.724, 113.791, -126.766, 55.289, 143.716]
  MoveL 200 to (321.91, 0, -0.55) mm, rotated rx -179.9 ry 0 rz -90 deg; joints [41.217, -71.756, 113.834, -126.753, 55.307, 143.716]
  MoveL 201 to (321.88, 0, -0.2) mm, rotated rx -179.9 ry 0 rz -90 deg; joints [41.226, -71.773, 113.856, -126.748, 55.316, 143.717]
  MoveL 202 to (321.83, 0, 0.15) mm, rotated rx -179.9 ry 0 rz -90 deg; joints [41.234, -71.79, 113.88, -126.743, 55.325, 143.719]
  MoveL 203 to (321.75, 0, 0.5) mm, rotated rx -179.9 ry 0 rz -90 deg; joints [41.241, -71.809, 113.905, -126.739, 55.333, 143.721]
  MoveL 204 to (321.66, 0, 0.84) mm, rotated rx -179.9 ry 0 rz -90 deg; joints [41.248, -71.828, 113.931, -126.736, 55.341, 143.724]
  MoveL 205 to (321.54, 0, 1.19) mm, rotated rx -179.9 ry 0 rz -90 deg; joints [41.255, -71.848, 113.959, -126.734, 55.349, 143.728]
  MoveL 206 to (321.4, 0, 1.54) mm, rotated rx -179.9 ry 0 rz -90 deg; joints [41.26, -71.869, 113.987, -126.733, 55.357, 143.732]
  MoveL 207 to (321.24, 0, 1.87) mm, rotated rx -179.9 ry 0 rz -90 deg; joints [41.264, -71.89, 114.015, -126.733, 55.364, 143.737]
  MoveL 208 to (321.07, 0, 2.19) mm, rotated rx -179.9 ry 0 rz -90 deg; joints [41.268, -71.911, 114.044, -126.734, 55.371, 143.742]
  MoveL 209 to (320.86, 0, 2.52) mm, rotated rx -179.9 ry 0 rz -90 deg; joints [41.271, -71.934, 114.075, -126.735, 55.377, 143.749]
  MoveL 210 to (320.63, 0, 2.85) mm, rotated rx -179.9 ry 0 rz -90 deg; joints [41.272, -71.957, 114.107, -126.738, 55.383, 143.756]
  MoveL 211 to (320.32, 0, 3.22) mm, rotated rx -179.9 ry 0 rz -90 deg; joints [41.273, -71.986, 114.146, -126.743, 55.39, 143.766]
  MoveL 212 to (319.96, 0, 3.6) mm, rotated rx -179.9 ry 0 rz -90 deg; joints [41.272, -72.017, 114.188, -126.751, 55.396, 143.777]
  MoveL 213 to (319.63, 0, 3.89) mm, rotated rx -179.9 ry 0 rz -90 deg; joints [41.27, -72.043, 114.224, -126.758, 55.4, 143.787]
  MoveL 214 to (319.29, 0, 4.15) mm, rotated rx -179.9 ry 0 rz -90 deg; joints [41.266, -72.068, 114.257, -126.766, 55.403, 143.798]
  MoveL 215 to (319.03, 0, 4.33) mm, rotated rx -179.9 ry 0 rz -90 deg; joints [41.263, -72.086, 114.282, -126.773, 55.405, 143.806]
  MoveL 216 to (318.71, 0, 4.52) mm, rotated rx -179.9 ry 0 rz -90 deg; joints [41.258, -72.107, 114.31, -126.782, 55.407, 143.816]
  MoveL 217 to (318.4, 0, 4.69) mm, rotated rx -179.9 ry 0 rz -90 deg; joints [41.252, -72.127, 114.337, -126.792, 55.408, 143.826]
  MoveL 218 to (318.08, 0, 4.84) mm, rotated rx -179.9 ry 0 rz -90 deg; joints [41.246, -72.145, 114.363, -126.801, 55.408, 143.836]
  MoveL 219 to (317.76, 0, 4.96) mm, rotated rx -179.9 ry 0 rz -90 deg; joints [41.24, -72.163, 114.387, -126.812, 55.408, 143.846]
  MoveL 220 to (317.45, 0, 5.07) mm, rotated rx -179.9 ry 0 rz -90 deg; joints [41.232, -72.18, 114.411, -126.822, 55.408, 143.856]
  MoveL 221 to (317.13, 0, 5.16) mm, rotated rx -179.9 ry 0 rz -90 deg; joints [41.224, -72.196, 114.433, -126.833, 55.407, 143.866]
  MoveL 222 to (316.82, 0, 5.23) mm, rotated rx -179.9 ry 0 rz -90 deg; joints [41.216, -72.212, 114.454, -126.844, 55.405, 143.876]
  MoveL 223 to (316.5, 0, 5.28) mm, rotated rx -179.9 ry 0 rz -90 deg; joints [41.207, -72.227, 114.474, -126.856, 55.403, 143.886]
  MoveL 224 to (316.15, 0, 5.32) mm, rotated rx -179.9 ry 0 rz -90 deg; joints [41.197, -72.242, 114.495, -126.869, 55.4, 143.897]
  MoveL 225 to (315.8, 0, 5.35) mm, rotated rx -179.9 ry 0 rz -90 deg; joints [41.186, -72.256, 114.515, -126.883, 55.397, 143.908]
  MoveL 226 to (315.11, 0, 5.35) mm, rotated rx -179.9 ry 0 rz -90 deg; joints [41.164, -72.284, 114.552, -126.911, 55.39, 143.93]
  MoveL 227 to (-302.56, 0, 5.35) mm, rotated rx -179.9 ry 0 rz -90 deg; joints [14.02, -90.531, 136.332, -160.507, 46.531, 166.759]
  MoveL 228 to (-303.26, 0, 5.35) mm, rotated rx -179.9 ry 0 rz -90 deg; joints [13.982, -90.542, 136.343, -160.558, 46.522, 166.793]
  MoveL 229 to (-303.6, 0, 5.33) mm, rotated rx -179.9 ry 0 rz -90 deg; joints [13.963, -90.546, 136.348, -160.584, 46.518, 166.811]
  MoveL 230 to (-303.95, 0, 5.29) mm, rotated rx -179.9 ry 0 rz -90 deg; joints [13.943, -90.549, 136.351, -160.61, 46.513, 166.829]
  MoveL 231 to (-304.3, 0, 5.23) mm, rotated rx -179.9 ry 0 rz -90 deg; joints [13.923, -90.551, 136.353, -160.637, 46.509, 166.847]
  MoveL 232 to (-304.65, 0, 5.15) mm, rotated rx -179.9 ry 0 rz -90 deg; joints [13.903, -90.552, 136.353, -160.664, 46.504, 166.865]
  MoveL 233 to (-305, 0, 5.05) mm, rotated rx -179.9 ry 0 rz -90 deg; joints [13.883, -90.55, 136.352, -160.692, 46.5, 166.884]
  MoveL 234 to (-305.35, 0, 4.92) mm, rotated rx -179.9 ry 0 rz -90 deg; joints [13.862, -90.548, 136.35, -160.72, 46.496, 166.903]
  MoveL 235 to (-305.64, 0, 4.8) mm, rotated rx -179.9 ry 0 rz -90 deg; joints [13.845, -90.545, 136.347, -160.743, 46.492, 166.919]
  MoveL 236 to (-305.93, 0, 4.67) mm, rotated rx -179.9 ry 0 rz -90 deg; joints [13.827, -90.54, 136.343, -160.767, 46.488, 166.935]
  MoveL 237 to (-306.22, 0, 4.51) mm, rotated rx -179.9 ry 0 rz -90 deg; joints [13.809, -90.534, 136.338, -160.791, 46.484, 166.951]
  MoveL 238 to (-306.51, 0, 4.33) mm, rotated rx -179.9 ry 0 rz -90 deg; joints [13.791, -90.527, 136.331, -160.816, 46.48, 166.968]
  MoveL 239 to (-306.92, 0, 4.05) mm, rotated rx -179.9 ry 0 rz -90 deg; joints [13.764, -90.515, 136.319, -160.851, 46.475, 166.992]
  MoveL 240 to (-307.32, 0, 3.71) mm, rotated rx -179.9 ry 0 rz -90 deg; joints [13.738, -90.499, 136.304, -160.887, 46.47, 167.017]
  MoveL 241 to (-307.55, 0, 3.5) mm, rotated rx -179.9 ry 0 rz -90 deg; joints [13.723, -90.488, 136.294, -160.908, 46.467, 167.031]
  MoveL 242 to (-307.77, 0, 3.26) mm, rotated rx -179.9 ry 0 rz -90 deg; joints [13.707, -90.476, 136.282, -160.928, 46.464, 167.045]
  MoveL 243 to (-307.96, 0, 3.04) mm, rotated rx -179.9 ry 0 rz -90 deg; joints [13.694, -90.464, 136.271, -160.947, 46.461, 167.057]
  MoveL 244 to (-308.14, 0, 2.82) mm, rotated rx -179.9 ry 0 rz -90 deg; joints [13.681, -90.452, 136.259, -160.964, 46.459, 167.069]
  MoveC 245 to (-308.98, 0, 2.34) mm, rotated rx -179.9 ry 0 rz -90 deg; joints [13.629, -90.434, 136.242, -161.035, 46.448, 167.117] to (-309.92, 0, 2.61) mm, rotated rx -179.9 ry 0 rz -90 deg; joints [13.581, -90.467, 136.274, -161.099, 46.437, 167.16]
  MoveL 246 to (-309.92, 0, 2.61) mm, rotated rx -179.9 ry 0 rz -90 deg; joints [13.581, -90.467, 136.274, -161.099, 46.437, 167.16]
  MoveL 247 to (-310.03, 0, 3.5) mm, rotated rx -179.9 ry 0 rz -90 deg; joints [13.587, -90.528, 136.334, -161.09, 46.436, 167.154]
  MoveL 248 to (-309.9, 0, 3.63) mm, rotated rx -179.9 ry 0 rz -90 deg; joints [13.596, -90.534, 136.34, -161.078, 46.438, 167.146]
  MoveL 249 to (-306.87, 0, 6.15) mm, rotated rx -179.9 ry 0 rz -90 deg; joints [13.796, -90.654, 136.454, -160.808, 46.478, 166.962]
  Set speed (50.0 mm/s)
  MoveL 250 to (-306.87, -4.73, 6.15) mm, rotated rx -179.9 ry 0 rz -90 deg; joints [13.798, -90.426, 136.63, -160.93, 46.861, 167.142]
  MoveC 251 to (-306.87, -5.63, 5.77) mm, rotated rx -179.9 ry 0 rz -90 deg; joints [13.793, -90.357, 136.639, -160.96, 46.933, 167.181] to (-306.87, -6, 4.88) mm, rotated rx -179.9 ry 0 rz -90 deg; joints [13.781, -90.279, 136.595, -160.987, 46.962, 167.207]
  MoveL 252 to (-306.87, -6, 4.88) mm, rotated rx -179.9 ry 0 rz -90 deg; joints [13.781, -90.279, 136.595, -160.987, 46.962, 167.207]
  Set speed (100.0 mm/s)
  MoveC 253 to (-307.24, -6, 3.98) mm, rotated rx -179.9 ry 0 rz -90 deg; joints [13.749, -90.226, 136.543, -161.03, 46.956, 167.237] to (-308.14, -6, 3.61) mm, rotated rx -179.9 ry 0 rz -90 deg; joints [13.694, -90.215, 136.534, -161.103, 46.945, 167.285]
  MoveL 254 to (-308.14, -6, 3.61) mm, rotated rx -179.9 ry 0 rz -90 deg; joints [13.694, -90.215, 136.534, -161.103, 46.945, 167.285]
  MoveL 255 to (-319.29, -6, 3.61) mm, rotated rx -179.9 ry 0 rz -90 deg; joints [13.083, -90.389, 136.71, -161.92, 46.813, 167.835]
  MoveL 256 to (-319.99, -6, 3.59) mm, rotated rx -179.9 ry 0 rz -90 deg; joints [13.045, -90.399, 136.72, -161.972, 46.805, 167.87]
  MoveL 257 to (-320.34, -6, 3.56) mm, rotated rx -179.9 ry 0 rz -90 deg; joints [13.025, -90.402, 136.723, -161.998, 46.801, 167.887]
  MoveL 258 to (-320.68, -6, 3.51) mm, rotated rx -179.9 ry 0 rz -90 deg; joints [13.005, -90.404, 136.725, -162.025, 46.797, 167.905]
  MoveL 259 to (-321.03, -6, 3.44) mm, rotated rx -179.9 ry 0 rz -90 deg; joints [12.985, -90.405, 136.726, -162.052, 46.793, 167.923]
  MoveL 260 to (-321.38, -6, 3.35) mm, rotated rx -179.9 ry 0 rz -90 deg; joints [12.965, -90.404, 136.725, -162.079, 46.789, 167.942]
  MoveL 261 to (-322.08, -6, 3.13) mm, rotated rx -179.9 ry 0 rz -90 deg; joints [12.924, -90.4, 136.722, -162.134, 46.781, 167.979]
  MoveL 262 to (-324.87, -6, 2.25) mm, rotated rx -179.9 ry 0 rz -90 deg; joints [12.759, -90.383, 136.707, -162.356, 46.748, 168.129]
  MoveL 263 to (-325.26, -6, 2.12) mm, rotated rx -179.9 ry 0 rz -90 deg; joints [12.736, -90.38, 136.704, -162.387, 46.744, 168.15]
  MoveL 264 to (-325.65, -6, 1.96) mm, rotated rx -179.9 ry 0 rz -90 deg; joints [12.713, -90.375, 136.7, -162.418, 46.739, 168.171]
  MoveL 265 to (-326.04, -6, 1.77) mm, rotated rx -179.9 ry 0 rz -90 deg; joints [12.689, -90.368, 136.693, -162.451, 46.735, 168.193]
  MoveL 266 to (-326.43, -6, 1.54) mm, rotated rx -179.9 ry 0 rz -90 deg; joints [12.665, -90.359, 136.685, -162.483, 46.73, 168.215]
  MoveL 267 to (-326.73, -6, 1.34) mm, rotated rx -179.9 ry 0 rz -90 deg; joints [12.645, -90.35, 136.676, -162.51, 46.727, 168.233]
  MoveL 268 to (-327.04, -6, 1.11) mm, rotated rx -179.9 ry 0 rz -90 deg; joints [12.625, -90.339, 136.665, -162.536, 46.723, 168.251]
  MoveL 269 to (-327.35, -6, 0.84) mm, rotated rx -179.9 ry 0 rz -90 deg; joints [12.605, -90.325, 136.653, -162.563, 46.719, 168.269]
  MoveL 270 to (-327.66, -6, 0.54) mm, rotated rx -179.9 ry 0 rz -90 deg; joints [12.585, -90.31, 136.638, -162.591, 46.716, 168.288]
  MoveL 271 to (-327.86, -6, 0.32) mm, rotated rx -179.9 ry 0 rz -90 deg; joints [12.571, -90.298, 136.626, -162.61, 46.713, 168.301]
  MoveL 272 to (-328.04, -6, 0.09) mm, rotated rx -179.9 ry 0 rz -90 deg; joints [12.558, -90.286, 136.615, -162.628, 46.711, 168.313]
  MoveL 273 to (-328.21, -6, -0.13) mm, rotated rx -179.9 ry 0 rz -90 deg; joints [12.546, -90.273, 136.603, -162.644, 46.709, 168.324]
  MoveL 274 to (-328.37, -6, -0.35) mm, rotated rx -179.9 ry 0 rz -90 deg; joints [12.534, -90.261, 136.59, -162.659, 46.707, 168.334]
  MoveL 275 to (-328.64, -6, -0.8) mm, rotated rx -179.9 ry 0 rz -90 deg; joints [12.514, -90.235, 136.565, -162.687, 46.704, 168.353]
  MoveL 276 to (-328.86, -6, -1.25) mm, rotated rx -179.9 ry 0 rz -90 deg; joints [12.497, -90.208, 136.539, -162.711, 46.701, 168.369]
  MoveL 277 to (-329, -6, -1.6) mm, rotated rx -179.9 ry 0 rz -90 deg; joints [12.484, -90.187, 136.519, -162.727, 46.699, 168.381]
  MoveL 278 to (-329.12, -6, -1.95) mm, rotated rx -179.9 ry 0 rz -90 deg; joints [12.473, -90.165, 136.498, -162.742, 46.697, 168.391]
  MoveL 279 to (-329.22, -6, -2.29) mm, rotated rx -179.9 ry 0 rz -90 deg; joints [12.464, -90.143, 136.477, -162.755, 46.696, 168.4]
  MoveL 280 to (-329.3, -6, -2.64) mm, rotated rx -179.9 ry 0 rz -90 deg; joints [12.455, -90.121, 136.455, -162.767, 46.695, 168.408]
  MoveL 281 to (-329.36, -6, -2.99) mm, rotated rx -179.9 ry 0 rz -90 deg; joints [12.448, -90.099, 136.433, -162.777, 46.694, 168.415]
  MoveL 282 to (-329.39, -6, -3.34) mm, rotated rx -179.9 ry 0 rz -90 deg; joints [12.442, -90.076, 136.411, -162.786, 46.693, 168.42]
  MoveL 283 to (-329.41, -6, -4.04) mm, rotated rx -179.9 ry 0 rz -90 deg; joints [12.432, -90.03, 136.366, -162.799, 46.692, 168.43]
  MoveL 284 to (-329.41, -6, -310.99) mm, rotated rx -179.9 ry 0 rz -90 deg; joints [9.546, -71.255, 114.238, -165.909, 42.91, 169.952]
  MoveL 285 to (-329.4, -6, -311.68) mm, rotated rx -179.9 ry 0 rz -90 deg; joints [9.542, -71.215, 114.183, -165.912, 42.895, 169.951]
  MoveL 286 to (-329.36, -6, -312.03) mm, rotated rx -179.9 ry 0 rz -90 deg; joints [9.541, -71.194, 114.154, -165.911, 42.887, 169.949]
  MoveL 287 to (-329.31, -6, -312.38) mm, rotated rx -179.9 ry 0 rz -90 deg; joints [9.54, -71.173, 114.126, -165.909, 42.88, 169.947]
  MoveL 288 to (-329.23, -6, -312.73) mm, rotated rx -179.9 ry 0 rz -90 deg; joints [9.541, -71.152, 114.097, -165.907, 42.872, 169.943]
  MoveL 289 to (-329.14, -6, -313.08) mm, rotated rx -179.9 ry 0 rz -90 deg; joints [9.543, -71.131, 114.068, -165.902, 42.865, 169.939]
  MoveL 290 to (-329.02, -6, -313.43) mm, rotated rx -179.9 ry 0 rz -90 deg; joints [9.545, -71.11, 114.039, -165.897, 42.858, 169.934]
  MoveL 291 to (-328.88, -6, -313.78) mm, rotated rx -179.9 ry 0 rz -90 deg; joints [9.548, -71.088, 114.009, -165.889, 42.85, 169.927]
  MoveL 292 to (-328.66, -6, -314.24) mm, rotated rx -179.9 ry 0 rz -90 deg; joints [9.555, -71.059, 113.969, -165.878, 42.841, 169.917]
  MoveL 293 to (-328.39, -6, -314.7) mm, rotated rx -179.9 ry 0 rz -90 deg; joints [9.563, -71.03, 113.929, -165.863, 42.832, 169.904]
  MoveL 294 to (-328.06, -6, -315.16) mm, rotated rx -179.9 ry 0 rz -90 deg; joints [9.574, -71, 113.887, -165.844, 42.823, 169.889]
  MoveL 295 to (-327.87, -6, -315.39) mm, rotated rx -179.9 ry 0 rz -90 deg; joints [9.58, -70.985, 113.866, -165.833, 42.818, 169.88]
  MoveL 296 to (-327.66, -6, -315.62) mm, rotated rx -179.9 ry 0 rz -90 deg; joints [9.587, -70.969, 113.845, -165.821, 42.814, 169.87]
  MoveL 297 to (-327.37, -6, -315.9) mm, rotated rx -179.9 ry 0 rz -90 deg; joints [9.597, -70.95, 113.819, -165.805, 42.808, 169.857]
  MoveL 298 to (-327.08, -6, -316.15) mm, rotated rx -179.9 ry 0 rz -90 deg; joints [9.608, -70.933, 113.795, -165.788, 42.804, 169.844]
  MoveL 299 to (-326.8, -6, -316.37) mm, rotated rx -179.9 ry 0 rz -90 deg; joints [9.618, -70.917, 113.773, -165.771, 42.8, 169.831]
  MoveL 300 to (-326.51, -6, -316.57) mm, rotated rx -179.9 ry 0 rz -90 deg; joints [9.629, -70.903, 113.754, -165.754, 42.797, 169.817]
  MoveL 301 to (-326.1, -6, -316.81) mm, rotated rx -179.9 ry 0 rz -90 deg; joints [9.645, -70.885, 113.729, -165.73, 42.793, 169.799]
  MoveL 302 to (-325.69, -6, -317.02) mm, rotated rx -179.9 ry 0 rz -90 deg; joints [9.661, -70.869, 113.706, -165.705, 42.79, 169.78]
  MoveL 303 to (-325.28, -6, -317.19) mm, rotated rx -179.9 ry 0 rz -90 deg; joints [9.677, -70.855, 113.687, -165.68, 42.787, 169.761]
  MoveL 304 to (-324.87, -6, -317.32) mm, rotated rx -179.9 ry 0 rz -90 deg; joints [9.693, -70.843, 113.671, -165.655, 42.786, 169.742]
  MoveL 305 to (-324.52, -6, -317.42) mm, rotated rx -179.9 ry 0 rz -90 deg; joints [9.708, -70.834, 113.658, -165.633, 42.785, 169.726]
  MoveL 306 to (-324.17, -6, -317.49) mm, rotated rx -179.9 ry 0 rz -90 deg; joints [9.722, -70.827, 113.648, -165.612, 42.785, 169.71]
  MoveL 307 to (-323.82, -6, -317.54) mm, rotated rx -179.9 ry 0 rz -90 deg; joints [9.736, -70.82, 113.639, -165.59, 42.785, 169.694]
  MoveL 308 to (-323.47, -6, -317.57) mm, rotated rx -179.9 ry 0 rz -90 deg; joints [9.751, -70.815, 113.631, -165.569, 42.785, 169.678]
  MoveL 309 to (-322.08, -6, -317.59) mm, rotated rx -179.9 ry 0 rz -90 deg; joints [9.81, -70.801, 113.61, -165.481, 42.79, 169.613]
  MoveL 310 to (324.87, -6, -317.59) mm, rotated rx -179.9 ry 0 rz -90 deg; joints [33.669, -56.318, 91.433, -130.018, 46.364, 141.417]
  MoveL 311 to (325.56, -6, -317.57) mm, rotated rx -179.9 ry 0 rz -90 deg; joints [33.69, -56.295, 91.395, -129.984, 46.368, 141.386]
  MoveL 312 to (325.91, -6, -317.53) mm, rotated rx -179.9 ry 0 rz -90 deg; joints [33.702, -56.284, 91.379, -129.968, 46.371, 141.371]
  MoveL 313 to (326.26, -6, -317.48) mm, rotated rx -179.9 ry 0 rz -90 deg; joints [33.713, -56.275, 91.364, -129.951, 46.375, 141.357]
  MoveL 314 to (326.61, -6, -317.4) mm, rotated rx -179.9 ry 0 rz -90 deg; joints [33.725, -56.267, 91.35, -129.934, 46.379, 141.342]
  MoveL 315 to (326.96, -6, -317.31) mm, rotated rx -179.9 ry 0 rz -90 deg; joints [33.738, -56.26, 91.339, -129.917, 46.384, 141.328]
  MoveL 316 to (327.31, -6, -317.19) mm, rotated rx -179.9 ry 0 rz -90 deg; joints [33.751, -56.254, 91.329, -129.9, 46.389, 141.315]
  MoveL 317 to (327.66, -6, -317.05) mm, rotated rx -179.9 ry 0 rz -90 deg; joints [33.764, -56.25, 91.321, -129.884, 46.396, 141.302]
  MoveL 318 to (328.1, -6, -316.83) mm, rotated rx -179.9 ry 0 rz -90 deg; joints [33.782, -56.246, 91.314, -129.862, 46.405, 141.286]
  MoveL 319 to (328.55, -6, -316.57) mm, rotated rx -179.9 ry 0 rz -90 deg; joints [33.801, -56.244, 91.311, -129.841, 46.416, 141.27]
  MoveL 320 to (328.84, -6, -316.37) mm, rotated rx -179.9 ry 0 rz -90 deg; joints [33.813, -56.244, 91.311, -129.827, 46.424, 141.261]
  MoveL 321 to (329.13, -6, -316.15) mm, rotated rx -179.9 ry 0 rz -90 deg; joints [33.827, -56.246, 91.313, -129.814, 46.432, 141.252]
  MoveL 322 to (329.41, -6, -315.9) mm, rotated rx -179.9 ry 0 rz -90 deg; joints [33.84, -56.249, 91.318, -129.8, 46.442, 141.244]
  MoveL 323 to (329.7, -6, -315.62) mm, rotated rx -179.9 ry 0 rz -90 deg; joints [33.855, -56.254, 91.325, -129.787, 46.453, 141.236]
  MoveL 324 to (329.91, -6, -315.38) mm, rotated rx -179.9 ry 0 rz -90 deg; joints [33.866, -56.258, 91.332, -129.776, 46.461, 141.231]
  MoveL 325 to (330.11, -6, -315.15) mm, rotated rx -179.9 ry 0 rz -90 deg; joints [33.877, -56.264, 91.341, -129.767, 46.47, 141.227]
  MoveL 326 to (330.28, -6, -314.91) mm, rotated rx -179.9 ry 0 rz -90 deg; joints [33.887, -56.27, 91.351, -129.759, 46.479, 141.223]
  MoveL 327 to (330.44, -6, -314.67) mm, rotated rx -179.9 ry 0 rz -90 deg; joints [33.896, -56.277, 91.361, -129.751, 46.487, 141.22]
  MoveL 328 to (330.71, -6, -314.22) mm, rotated rx -179.9 ry 0 rz -90 deg; joints [33.913, -56.291, 91.384, -129.739, 46.503, 141.217]
  MoveL 329 to (330.92, -6, -313.78) mm, rotated rx -179.9 ry 0 rz -90 deg; joints [33.929, -56.307, 91.409, -129.729, 46.519, 141.215]
  MoveL 330 to (331.06, -6, -313.43) mm, rotated rx -179.9 ry 0 rz -90 deg; joints [33.94, -56.32, 91.429, -129.723, 46.531, 141.215]
  MoveL 331 to (331.18, -6, -313.08) mm, rotated rx -179.9 ry 0 rz -90 deg; joints [33.951, -56.334, 91.452, -129.717, 46.543, 141.216]
  MoveL 332 to (331.28, -6, -312.73) mm, rotated rx -179.9 ry 0 rz -90 deg; joints [33.961, -56.348, 91.475, -129.713, 46.555, 141.218]
  MoveL 333 to (331.35, -6, -312.38) mm, rotated rx -179.9 ry 0 rz -90 deg; joints [33.97, -56.364, 91.5, -129.71, 46.567, 141.221]
  MoveL 334 to (331.4, -6, -312.03) mm, rotated rx -179.9 ry 0 rz -90 deg; joints [33.979, -56.38, 91.526, -129.707, 46.578, 141.225]
  MoveL 335 to (331.44, -6, -311.68) mm, rotated rx -179.9 ry 0 rz -90 deg; joints [33.987, -56.397, 91.552, -129.706, 46.59, 141.23]
  MoveL 336 to (331.45, -6, -310.99) mm, rotated rx -179.9 ry 0 rz -90 deg; joints [34.002, -56.432, 91.609, -129.706, 46.613, 141.242]
  MoveL 337 to (331.45, -6, -4.04) mm, rotated rx -179.9 ry 0 rz -90 deg; joints [41.43, -71.013, 113.294, -126.657, 55.555, 143.8]
  MoveL 338 to (331.45, -6, -2.64) mm, rotated rx -179.9 ry 0 rz -90 deg; joints [41.469, -71.075, 113.379, -126.631, 55.592, 143.8]
  MoveL 339 to (331.44, -6, -2.29) mm, rotated rx -179.9 ry 0 rz -90 deg; joints [41.479, -71.091, 113.401, -126.625, 55.601, 143.801]
  MoveL 340 to (331.4, -6, -1.95) mm, rotated rx -179.9 ry 0 rz -90 deg; joints [41.488, -71.108, 113.424, -126.62, 55.61, 143.802]
  MoveL 341 to (331.35, -6, -1.6) mm, rotated rx -179.9 ry 0 rz -90 deg; joints [41.496, -71.125, 113.448, -126.615, 55.619, 143.804]
  MoveL 342 to (331.28, -6, -1.25) mm, rotated rx -179.9 ry 0 rz -90 deg; joints [41.504, -71.144, 113.473, -126.611, 55.628, 143.806]
  MoveL 343 to (331.14, -6, -0.76) mm, rotated rx -179.9 ry 0 rz -90 deg; joints [41.513, -71.171, 113.509, -126.608, 55.639, 143.811]
  MoveL 344 to (330.96, -6, -0.28) mm, rotated rx -179.9 ry 0 rz -90 deg; joints [41.521, -71.199, 113.549, -126.606, 55.65, 143.817]
  MoveL 345 to (330.73, -6, 0.21) mm, rotated rx -179.9 ry 0 rz -90 deg; joints [41.528, -71.23, 113.59, -126.605, 55.661, 143.824]
  MoveL 346 to (330.59, -6, 0.45) mm, rotated rx -179.9 ry 0 rz -90 deg; joints [41.53, -71.246, 113.612, -126.606, 55.666, 143.829]
  MoveL 347 to (330.44, -6, 0.69) mm, rotated rx -179.9 ry 0 rz -90 deg; joints [41.532, -71.262, 113.635, -126.607, 55.671, 143.834]
  MoveL 348 to (330.15, -6, 1.12) mm, rotated rx -179.9 ry 0 rz -90 deg; joints [41.535, -71.293, 113.677, -126.611, 55.679, 143.843]
  MoveL 349 to (329.98, -6, 1.33) mm, rotated rx -179.9 ry 0 rz -90 deg; joints [41.536, -71.309, 113.699, -126.614, 55.683, 143.849]
  MoveL 350 to (329.79, -6, 1.54) mm, rotated rx -179.9 ry 0 rz -90 deg; joints [41.536, -71.325, 113.722, -126.617, 55.687, 143.855]
  MoveL 351 to (329.52, -6, 1.82) mm, rotated rx -179.9 ry 0 rz -90 deg; joints [41.535, -71.348, 113.753, -126.623, 55.691, 143.863]
  MoveL 352 to (329.26, -6, 2.06) mm, rotated rx -179.9 ry 0 rz -90 deg; joints [41.533, -71.369, 113.782, -126.628, 55.695, 143.872]
  MoveL 353 to (328.99, -6, 2.28) mm, rotated rx -179.9 ry 0 rz -90 deg; joints [41.531, -71.389, 113.809, -126.635, 55.698, 143.88]
  MoveL 354 to (328.72, -6, 2.47) mm, rotated rx -179.9 ry 0 rz -90 deg; joints [41.528, -71.408, 113.835, -126.642, 55.701, 143.889]
  MoveL 355 to (328.46, -6, 2.65) mm, rotated rx -179.9 ry 0 rz -90 deg; joints [41.524, -71.426, 113.86, -126.649, 55.703, 143.898]
  MoveL 356 to (328.19, -6, 2.81) mm, rotated rx -179.9 ry 0 rz -90 deg; joints [41.52, -71.443, 113.884, -126.657, 55.704, 143.906]
  MoveL 357 to (327.92, -6, 2.95) mm, rotated rx -179.9 ry 0 rz -90 deg; joints [41.516, -71.46, 113.907, -126.664, 55.705, 143.915]
  MoveL 358 to (327.66, -6, 3.07) mm, rotated rx -179.9 ry 0 rz -90 deg; joints [41.511, -71.476, 113.929, -126.673, 55.706, 143.923]
  MoveL 359 to (327.31, -6, 3.21) mm, rotated rx -179.9 ry 0 rz -90 deg; joints [41.503, -71.496, 113.956, -126.684, 55.706, 143.934]
  MoveL 360 to (326.96, -6, 3.33) mm, rotated rx -179.9 ry 0 rz -90 deg; joints [41.495, -71.514, 113.982, -126.695, 55.705, 143.946]
  MoveL 361 to (326.61, -6, 3.42) mm, rotated rx -179.9 ry 0 rz -90 deg; joints [41.487, -71.532, 114.007, -126.708, 55.704, 143.957]
  MoveL 362 to (326.26, -6, 3.5) mm, rotated rx -179.9 ry 0 rz -90 deg; joints [41.478, -71.549, 114.03, -126.72, 55.703, 143.968]
  MoveL 363 to (325.91, -6, 3.55) mm, rotated rx -179.9 ry 0 rz -90 deg; joints [41.468, -71.565, 114.052, -126.733, 55.701, 143.979]
  MoveL 364 to (325.56, -6, 3.59) mm, rotated rx -179.9 ry 0 rz -90 deg; joints [41.458, -71.58, 114.073, -126.746, 55.698, 143.99]
  MoveL 365 to (324.87, -6, 3.61) mm, rotated rx -179.9 ry 0 rz -90 deg; joints [41.436, -71.608, 114.111, -126.774, 55.692, 144.012]
  MoveL 366 to (319.99, -6, 3.61) mm, rotated rx -179.9 ry 0 rz -90 deg; joints [41.277, -71.797, 114.373, -126.969, 55.642, 144.168]
  MoveL 367 to (319.81, -6, 3.73) mm, rotated rx -179.9 ry 0 rz -90 deg; joints [41.275, -71.809, 114.39, -126.973, 55.643, 144.174]
  MoveL 368 to (319.64, -6, 3.88) mm, rotated rx -179.9 ry 0 rz -90 deg; joints [41.273, -71.822, 114.409, -126.978, 55.646, 144.179]
  MoveL 369 to (319.29, -6, 4.15) mm, rotated rx -179.9 ry 0 rz -90 deg; joints [41.27, -71.848, 114.444, -126.986, 55.649, 144.19]
  MoveL 370 to (319.03, -6, 4.33) mm, rotated rx -179.9 ry 0 rz -90 deg; joints [41.266, -71.866, 114.468, -126.993, 55.651, 144.199]
  MoveL 371 to (318.71, -6, 4.52) mm, rotated rx -179.9 ry 0 rz -90 deg; joints [41.261, -71.887, 114.497, -127.002, 55.653, 144.209]
  MoveL 372 to (318.4, -6, 4.69) mm, rotated rx -179.9 ry 0 rz -90 deg; joints [41.256, -71.906, 114.524, -127.011, 55.654, 144.219]
  MoveL 373 to (318.08, -6, 4.84) mm, rotated rx -179.9 ry 0 rz -90 deg; joints [41.25, -71.925, 114.549, -127.021, 55.655, 144.229]
  MoveL 374 to (317.76, -6, 4.96) mm, rotated rx -179.9 ry 0 rz -90 deg; joints [41.243, -71.943, 114.574, -127.031, 55.655, 144.239]
  MoveL 375 to (317.45, -6, 5.07) mm, rotated rx -179.9 ry 0 rz -90 deg; joints [41.236, -71.96, 114.597, -127.042, 55.654, 144.249]
  MoveL 376 to (317.13, -6, 5.16) mm, rotated rx -179.9 ry 0 rz -90 deg; joints [41.228, -71.976, 114.619, -127.053, 55.653, 144.259]
  MoveL 377 to (316.82, -6, 5.23) mm, rotated rx -179.9 ry 0 rz -90 deg; joints [41.22, -71.991, 114.64, -127.064, 55.652, 144.269]
  MoveL 378 to (316.5, -6, 5.28) mm, rotated rx -179.9 ry 0 rz -90 deg; joints [41.211, -72.006, 114.66, -127.076, 55.65, 144.279]
  MoveL 379 to (316.15, -6, 5.32) mm, rotated rx -179.9 ry 0 rz -90 deg; joints [41.201, -72.021, 114.682, -127.089, 55.647, 144.29]
  MoveL 380 to (315.8, -6, 5.35) mm, rotated rx -179.9 ry 0 rz -90 deg; joints [41.19, -72.036, 114.701, -127.103, 55.644, 144.301]
  MoveL 381 to (315.11, -6, 5.35) mm, rotated rx -179.9 ry 0 rz -90 deg; joints [41.167, -72.063, 114.739, -127.13, 55.637, 144.323]
  MoveL 382 to (-302.56, -6, 5.35) mm, rotated rx -179.9 ry 0 rz -90 deg; joints [14.023, -90.241, 136.555, -160.664, 47.015, 166.99]
  MoveL 383 to (-303.26, -6, 5.35) mm, rotated rx -179.9 ry 0 rz -90 deg; joints [13.985, -90.252, 136.566, -160.715, 47.007, 167.024]
  MoveL 384 to (-303.6, -6, 5.33) mm, rotated rx -179.9 ry 0 rz -90 deg; joints [13.965, -90.257, 136.571, -160.74, 47.002, 167.042]
  MoveL 385 to (-303.95, -6, 5.29) mm, rotated rx -179.9 ry 0 rz -90 deg; joints [13.946, -90.26, 136.574, -160.767, 46.998, 167.059]
  MoveL 386 to (-304.3, -6, 5.23) mm, rotated rx -179.9 ry 0 rz -90 deg; joints [13.926, -90.262, 136.576, -160.793, 46.994, 167.077]
  MoveL 387 to (-304.65, -6, 5.15) mm, rotated rx -179.9 ry 0 rz -90 deg; joints [13.906, -90.262, 136.577, -160.82, 46.989, 167.095]
  MoveL 388 to (-305, -6, 5.05) mm, rotated rx -179.9 ry 0 rz -90 deg; joints [13.885, -90.261, 136.576, -160.847, 46.985, 167.113]
  MoveL 389 to (-305.35, -6, 4.92) mm, rotated rx -179.9 ry 0 rz -90 deg; joints [13.865, -90.258, 136.573, -160.875, 46.981, 167.132]
  MoveL 390 to (-305.64, -6, 4.8) mm, rotated rx -179.9 ry 0 rz -90 deg; joints [13.847, -90.255, 136.57, -160.898, 46.977, 167.148]
  MoveL 391 to (-305.93, -6, 4.67) mm, rotated rx -179.9 ry 0 rz -90 deg; joints [13.829, -90.251, 136.566, -160.922, 46.973, 167.164]
  MoveL 392 to (-306.22, -6, 4.51) mm, rotated rx -179.9 ry 0 rz -90 deg; joints [13.811, -90.245, 136.561, -160.946, 46.969, 167.18]
  MoveL 393 to (-306.51, -6, 4.33) mm, rotated rx -179.9 ry 0 rz -90 deg; joints [13.793, -90.238, 136.554, -160.971, 46.966, 167.196]
  MoveL 394 to (-306.92, -6, 4.05) mm, rotated rx -179.9 ry 0 rz -90 deg; joints [13.767, -90.225, 136.542, -161.006, 46.96, 167.22]
  MoveL 395 to (-307.32, -6, 3.71) mm, rotated rx -179.9 ry 0 rz -90 deg; joints [13.74, -90.209, 136.527, -161.041, 46.955, 167.244]
  MoveL 396 to (-307.53, -6, 3.61) mm, rotated rx -179.9 ry 0 rz -90 deg; joints [13.728, -90.206, 136.524, -161.058, 46.952, 167.255]
  MoveL 397 to (-308.14, -6, 3.61) mm, rotated rx -179.9 ry 0 rz -90 deg; joints [13.694, -90.215, 136.534, -161.103, 46.945, 167.285]
  MoveC 398 to (-309.41, -6, 4.88) mm, rotated rx -179.9 ry 0 rz -90 deg; joints [13.642, -90.32, 136.636, -161.172, 46.931, 167.331] to (-308.14, -6, 6.15) mm, rotated rx -179.9 ry 0 rz -90 deg; joints [13.729, -90.384, 136.698, -161.056, 46.948, 167.253]
  MoveL 399 to (-308.14, -6, 6.15) mm, rotated rx -179.9 ry 0 rz -90 deg; joints [13.729, -90.384, 136.698, -161.056, 46.948, 167.253]
  MoveL 400 to (-306.87, -6, 6.15) mm, rotated rx -179.9 ry 0 rz -90 deg; joints [13.798, -90.364, 136.677, -160.963, 46.964, 167.19]
  Set speed (50.0 mm/s)
  MoveL 401 to (-306.87, -8.26, 6.15) mm, rotated rx -179.9 ry 0 rz -90 deg; joints [13.799, -90.254, 136.761, -161.02, 47.147, 167.276]
  MoveC 402 to (-306.87, -9.15, 5.77) mm, rotated rx -179.9 ry 0 rz -90 deg; joints [13.794, -90.185, 136.769, -161.05, 47.219, 167.314] to (-306.87, -9.52, 4.88) mm, rotated rx -179.9 ry 0 rz -90 deg; joints [13.782, -90.107, 136.725, -161.076, 47.248, 167.34]
  MoveL 403 to (-306.87, -9.52, 4.88) mm, rotated rx -179.9 ry 0 rz -90 deg; joints [13.782, -90.107, 136.725, -161.076, 47.248, 167.34]
  Set speed (100.0 mm/s)
  MoveC 404 to (-307.24, -9.53, 3.98) mm, rotated rx -179.9 ry 0 rz -90 deg; joints [13.75, -90.054, 136.673, -161.119, 47.242, 167.369] to (-308.14, -9.52, 3.61) mm, rotated rx -179.9 ry 0 rz -90 deg; joints [13.696, -90.043, 136.663, -161.191, 47.231, 167.417]
  MoveL 405 to (-308.14, -9.52, 3.61) mm, rotated rx -179.9 ry 0 rz -90 deg; joints [13.696, -90.043, 136.663, -161.191, 47.231, 167.417]
  MoveL 406 to (-319.29, -9.52, 3.61) mm, rotated rx -179.9 ry 0 rz -90 deg; joints [13.085, -90.217, 136.84, -162.006, 47.101, 167.962]
  MoveL 407 to (-319.99, -9.52, 3.59) mm, rotated rx -179.9 ry 0 rz -90 deg; joints [13.046, -90.227, 136.85, -162.057, 47.093, 167.996]
  MoveL 408 to (-320.34, -9.53, 3.56) mm, rotated rx -179.9 ry 0 rz -90 deg; joints [13.027, -90.23, 136.853, -162.083, 47.089, 168.014]
  MoveL 409 to (-320.68, -9.53, 3.51) mm, rotated rx -179.9 ry 0 rz -90 deg; joints [13.007, -90.232, 136.855, -162.11, 47.085, 168.031]
  MoveL 410 to (-321.03, -9.53, 3.44) mm, rotated rx -179.9 ry 0 rz -90 deg; joints [12.987, -90.232, 136.856, -162.137, 47.081, 168.049]
  MoveL 411 to (-321.38, -9.52, 3.35) mm, rotated rx -179.9 ry 0 rz -90 deg; joints [12.966, -90.231, 136.855, -162.164, 47.077, 168.068]
  MoveL 412 to (-322.08, -9.52, 3.13) mm, rotated rx -179.9 ry 0 rz -90 deg; joints [12.925, -90.227, 136.852, -162.219, 47.069, 168.105]
  MoveL 413 to (-327.09, -9.53, 1.54) mm, rotated rx -179.9 ry 0 rz -90 deg; joints [12.629, -90.196, 136.825, -162.615, 47.012, 168.371]
  MoveL 414 to (-327.37, -9.53, 1.44) mm, rotated rx -179.9 ry 0 rz -90 deg; joints [12.613, -90.193, 136.822, -162.638, 47.008, 168.386]
  MoveL 415 to (-327.66, -9.53, 1.33) mm, rotated rx -179.9 ry 0 rz -90 deg; joints [12.596, -90.19, 136.819, -162.661, 47.005, 168.401]
  MoveL 416 to (-328, -9.53, 1.16) mm, rotated rx -179.9 ry 0 rz -90 deg; joints [12.575, -90.184, 136.813, -162.689, 47.001, 168.42]
  MoveL 417 to (-328.35, -9.53, 0.97) mm, rotated rx -179.9 ry 0 rz -90 deg; joints [12.553, -90.176, 136.806, -162.718, 46.997, 168.44]
  MoveL 418 to (-328.7, -9.53, 0.74) mm, rotated rx -179.9 ry 0 rz -90 deg; joints [12.531, -90.166, 136.796, -162.748, 46.993, 168.46]
  MoveL 419 to (-329.05, -9.53, 0.48) mm, rotated rx -179.9 ry 0 rz -90 deg; joints [12.509, -90.154, 136.785, -162.778, 46.989, 168.48]
  MoveL 420 to (-329.25, -9.52, 0.32) mm, rotated rx -179.9 ry 0 rz -90 deg; joints [12.495, -90.146, 136.777, -162.796, 46.987, 168.492]
  MoveL 421 to (-329.46, -9.53, 0.13) mm, rotated rx -179.9 ry 0 rz -90 deg; joints [12.482, -90.136, 136.768, -162.814, 46.984, 168.504]
  MoveL 422 to (-329.67, -9.52, -0.08) mm, rotated rx -179.9 ry 0 rz -90 deg; joints [12.468, -90.126, 136.757, -162.833, 46.982, 168.517]
  MoveL 423 to (-329.86, -9.52, -0.29) mm, rotated rx -179.9 ry 0 rz -90 deg; joints [12.455, -90.114, 136.747, -162.851, 46.98, 168.529]
  MoveL 424 to (-330.18, -9.53, -0.67) mm, rotated rx -179.9 ry 0 rz -90 deg; joints [12.433, -90.093, 136.726, -162.88, 46.976, 168.549]
  MoveL 425 to (-330.44, -9.52, -1.06) mm, rotated rx -179.9 ry 0 rz -90 deg; joints [12.413, -90.071, 136.705, -162.907, 46.972, 168.567]
  MoveL 426 to (-330.56, -9.52, -1.25) mm, rotated rx -179.9 ry 0 rz -90 deg; joints [12.404, -90.06, 136.694, -162.918, 46.971, 168.575]
  MoveL 427 to (-330.75, -9.52, -1.6) mm, rotated rx -179.9 ry 0 rz -90 deg; joints [12.39, -90.04, 136.674, -162.938, 46.969, 168.588]
  MoveL 428 to (-330.92, -9.53, -1.95) mm, rotated rx -179.9 ry 0 rz -90 deg; joints [12.376, -90.019, 136.654, -162.956, 46.966, 168.601]
  MoveL 429 to (-331.06, -9.53, -2.29) mm, rotated rx -179.9 ry 0 rz -90 deg; joints [12.364, -89.998, 136.633, -162.972, 46.964, 168.612]
  MoveL 430 to (-331.18, -9.53, -2.64) mm, rotated rx -179.9 ry 0 rz -90 deg; joints [12.354, -89.976, 136.612, -162.987, 46.963, 168.621]
  MoveL 431 to (-331.27, -9.53, -2.99) mm, rotated rx -179.9 ry 0 rz -90 deg; joints [12.344, -89.954, 136.591, -163, 46.961, 168.63]
  MoveL 432 to (-331.34, -9.52, -3.34) mm, rotated rx -179.9 ry 0 rz -90 deg; joints [12.336, -89.932, 136.569, -163.011, 46.96, 168.638]
  MoveL 433 to (-331.4, -9.53, -3.69) mm, rotated rx -179.9 ry 0 rz -90 deg; joints [12.329, -89.91, 136.547, -163.021, 46.959, 168.644]
  MoveL 434 to (-331.43, -9.52, -4.04) mm, rotated rx -179.9 ry 0 rz -90 deg; joints [12.323, -89.887, 136.525, -163.029, 46.958, 168.65]
  MoveL 435 to (-331.45, -9.53, -6.83) mm, rotated rx -179.9 ry 0 rz -90 deg; joints [12.288, -89.702, 136.343, -163.076, 46.954, 168.682]
  MoveL 436 to (-331.45, -9.52, -310.99) mm, rotated rx -179.9 ry 0 rz -90 deg; joints [9.46, -71.144, 114.374, -166.097, 43.134, 170.129]
  MoveL 437 to (-331.43, -9.52, -311.68) mm, rotated rx -179.9 ry 0 rz -90 deg; joints [9.456, -71.104, 114.318, -166.1, 43.119, 170.128]
  MoveL 438 to (-331.4, -9.53, -312.03) mm, rotated rx -179.9 ry 0 rz -90 deg; joints [9.455, -71.083, 114.29, -166.099, 43.111, 170.126]
  MoveL 439 to (-331.34, -9.53, -312.38) mm, rotated rx -179.9 ry 0 rz -90 deg; joints [9.454, -71.062, 114.261, -166.097, 43.103, 170.124]
  MoveL 440 to (-331.27, -9.53, -312.73) mm, rotated rx -179.9 ry 0 rz -90 deg; joints [9.455, -71.041, 114.232, -166.094, 43.096, 170.12]
  MoveL 441 to (-331.17, -9.52, -313.08) mm, rotated rx -179.9 ry 0 rz -90 deg; joints [9.457, -71.02, 114.203, -166.09, 43.088, 170.116]
  MoveL 442 to (-331.06, -9.53, -313.43) mm, rotated rx -179.9 ry 0 rz -90 deg; joints [9.459, -70.999, 114.174, -166.085, 43.081, 170.11]
  MoveL 443 to (-330.92, -9.52, -313.78) mm, rotated rx -179.9 ry 0 rz -90 deg; joints [9.463, -70.977, 114.144, -166.077, 43.074, 170.104]
  MoveL 444 to (-330.7, -9.53, -314.22) mm, rotated rx -179.9 ry 0 rz -90 deg; joints [9.469, -70.95, 114.106, -166.066, 43.065, 170.094]
  MoveL 445 to (-330.44, -9.52, -314.66) mm, rotated rx -179.9 ry 0 rz -90 deg; joints [9.476, -70.921, 114.067, -166.052, 43.056, 170.082]
  MoveL 446 to (-330.11, -9.53, -315.14) mm, rotated rx -179.9 ry 0 rz -90 deg; joints [9.487, -70.891, 114.025, -166.033, 43.046, 170.067]
  MoveL 447 to (-329.91, -9.53, -315.38) mm, rotated rx -179.9 ry 0 rz -90 deg; joints [9.494, -70.875, 114.003, -166.022, 43.041, 170.058]
  MoveL 448 to (-329.7, -9.52, -315.61) mm, rotated rx -179.9 ry 0 rz -90 deg; joints [9.501, -70.859, 113.981, -166.01, 43.037, 170.048]
  MoveL 449 to (-329.41, -9.53, -315.9) mm, rotated rx -179.9 ry 0 rz -90 deg; joints [9.512, -70.84, 113.954, -165.993, 43.032, 170.035]
  MoveL 450 to (-329.12, -9.53, -316.15) mm, rotated rx -179.9 ry 0 rz -90 deg; joints [9.522, -70.823, 113.93, -165.976, 43.027, 170.021]
  MoveL 451 to (-328.83, -9.53, -316.37) mm, rotated rx -179.9 ry 0 rz -90 deg; joints [9.533, -70.807, 113.909, -165.959, 43.023, 170.008]
  MoveL 452 to (-328.55, -9.52, -316.57) mm, rotated rx -179.9 ry 0 rz -90 deg; joints [9.544, -70.793, 113.889, -165.942, 43.02, 169.995]
  MoveL 453 to (-328.1, -9.52, -316.83) mm, rotated rx -179.9 ry 0 rz -90 deg; joints [9.561, -70.773, 113.862, -165.916, 43.015, 169.975]
  MoveL 454 to (-327.66, -9.53, -317.05) mm, rotated rx -179.9 ry 0 rz -90 deg; joints [9.578, -70.756, 113.839, -165.889, 43.012, 169.954]
  MoveL 455 to (-327.31, -9.53, -317.19) mm, rotated rx -179.9 ry 0 rz -90 deg; joints [9.592, -70.745, 113.822, -165.868, 43.01, 169.938]
  MoveL 456 to (-326.96, -9.52, -317.31) mm, rotated rx -179.9 ry 0 rz -90 deg; joints [9.606, -70.735, 113.808, -165.847, 43.008, 169.922]
  MoveL 457 to (-326.61, -9.52, -317.4) mm, rotated rx -179.9 ry 0 rz -90 deg; joints [9.62, -70.726, 113.796, -165.826, 43.008, 169.906]
  MoveL 458 to (-326.26, -9.53, -317.48) mm, rotated rx -179.9 ry 0 rz -90 deg; joints [9.634, -70.718, 113.785, -165.804, 43.007, 169.89]
  MoveL 459 to (-325.91, -9.52, -317.53) mm, rotated rx -179.9 ry 0 rz -90 deg; joints [9.649, -70.711, 113.776, -165.783, 43.007, 169.874]
  MoveL 460 to (-325.56, -9.52, -317.57) mm, rotated rx -179.9 ry 0 rz -90 deg; joints [9.663, -70.706, 113.768, -165.761, 43.007, 169.859]
  MoveL 461 to (-324.87, -9.52, -317.59) mm, rotated rx -179.9 ry 0 rz -90 deg; joints [9.693, -70.698, 113.757, -165.718, 43.01, 169.827]
  MoveL 462 to (324.87, -9.53, -317.59) mm, rotated rx -179.9 ry 0 rz -90 deg; joints [33.671, -56.218, 91.538, -130.166, 46.498, 141.633]
  MoveL 463 to (325.56, -9.52, -317.57) mm, rotated rx -179.9 ry 0 rz -90 deg; joints [33.692, -56.195, 91.501, -130.132, 46.501, 141.602]
  MoveL 464 to (325.91, -9.53, -317.53) mm, rotated rx -179.9 ry 0 rz -90 deg; joints [33.703, -56.185, 91.484, -130.115, 46.504, 141.587]
  MoveL 465 to (326.26, -9.53, -317.48) mm, rotated rx -179.9 ry 0 rz -90 deg; joints [33.715, -56.176, 91.469, -130.099, 46.508, 141.573]
  MoveL 466 to (326.61, -9.53, -317.4) mm, rotated rx -179.9 ry 0 rz -90 deg; joints [33.727, -56.168, 91.456, -130.082, 46.512, 141.558]
  MoveL 467 to (326.96, -9.53, -317.31) mm, rotated rx -179.9 ry 0 rz -90 deg; joints [33.739, -56.161, 91.444, -130.065, 46.517, 141.544]
  MoveL 468 to (327.31, -9.52, -317.19) mm, rotated rx -179.9 ry 0 rz -90 deg; joints [33.752, -56.155, 91.435, -130.048, 46.522, 141.531]
  MoveL 469 to (327.66, -9.52, -317.05) mm, rotated rx -179.9 ry 0 rz -90 deg; joints [33.766, -56.15, 91.427, -130.032, 46.529, 141.518]
  MoveL 470 to (328.1, -9.53, -316.83) mm, rotated rx -179.9 ry 0 rz -90 deg; joints [33.784, -56.146, 91.42, -130.01, 46.538, 141.502]
  MoveL 471 to (328.55, -9.53, -316.57) mm, rotated rx -179.9 ry 0 rz -90 deg; joints [33.802, -56.144, 91.416, -129.989, 46.549, 141.487]
  MoveL 472 to (328.84, -9.53, -316.37) mm, rotated rx -179.9 ry 0 rz -90 deg; joints [33.815, -56.145, 91.417, -129.975, 46.556, 141.477]
  MoveL 473 to (329.13, -9.52, -316.15) mm, rotated rx -179.9 ry 0 rz -90 deg; joints [33.828, -56.146, 91.419, -129.962, 46.565, 141.469]
  MoveL 474 to (329.41, -9.52, -315.9) mm, rotated rx -179.9 ry 0 rz -90 deg; joints [33.842, -56.149, 91.423, -129.948, 46.575, 141.46]
  MoveL 475 to (329.7, -9.52, -315.62) mm, rotated rx -179.9 ry 0 rz -90 deg; joints [33.856, -56.154, 91.431, -129.934, 46.585, 141.453]
  MoveL 476 to (329.91, -9.53, -315.38) mm, rotated rx -179.9 ry 0 rz -90 deg; joints [33.867, -56.159, 91.438, -129.924, 46.594, 141.447]
  MoveL 477 to (330.11, -9.52, -315.15) mm, rotated rx -179.9 ry 0 rz -90 deg; joints [33.878, -56.164, 91.447, -129.915, 46.603, 141.443]
  MoveL 478 to (330.28, -9.52, -314.91) mm, rotated rx -179.9 ry 0 rz -90 deg; joints [33.888, -56.171, 91.457, -129.907, 46.611, 141.439]
  MoveL 479 to (330.44, -9.53, -314.67) mm, rotated rx -179.9 ry 0 rz -90 deg; joints [33.898, -56.177, 91.467, -129.899, 46.62, 141.436]
  MoveL 480 to (330.71, -9.52, -314.22) mm, rotated rx -179.9 ry 0 rz -90 deg; joints [33.915, -56.191, 91.489, -129.887, 46.636, 141.433]
  MoveL 481 to (330.92, -9.53, -313.78) mm, rotated rx -179.9 ry 0 rz -90 deg; joints [33.931, -56.207, 91.514, -129.877, 46.651, 141.431]
  MoveL 482 to (331.06, -9.53, -313.43) mm, rotated rx -179.9 ry 0 rz -90 deg; joints [33.942, -56.22, 91.535, -129.87, 46.664, 141.431]
  MoveL 483 to (331.18, -9.53, -313.08) mm, rotated rx -179.9 ry 0 rz -90 deg; joints [33.953, -56.234, 91.557, -129.865, 46.676, 141.433]
  MoveL 484 to (331.28, -9.53, -312.73) mm, rotated rx -179.9 ry 0 rz -90 deg; joints [33.962, -56.249, 91.581, -129.861, 46.687, 141.435]
  MoveL 485 to (331.35, -9.53, -312.38) mm, rotated rx -179.9 ry 0 rz -90 deg; joints [33.972, -56.264, 91.606, -129.857, 46.699, 141.438]
  MoveL 486 to (331.4, -9.53, -312.03) mm, rotated rx -179.9 ry 0 rz -90 deg; joints [33.981, -56.28, 91.631, -129.855, 46.711, 141.441]
  MoveL 487 to (331.44, -9.52, -311.68) mm, rotated rx -179.9 ry 0 rz -90 deg; joints [33.989, -56.297, 91.658, -129.854, 46.722, 141.446]
  MoveL 488 to (331.45, -9.53, -310.99) mm, rotated rx -179.9 ry 0 rz -90 deg; joints [34.003, -56.332, 91.715, -129.853, 46.745, 141.458]
  MoveL 489 to (331.45, -9.53, -4.04) mm, rotated rx -179.9 ry 0 rz -90 deg; joints [41.432, -70.884, 113.402, -126.785, 55.698, 144.028]
  MoveL 490 to (331.45, -9.52, -2.64) mm, rotated rx -179.9 ry 0 rz -90 deg; joints [41.472, -70.946, 113.486, -126.759, 55.735, 144.029]
  MoveL 491 to (331.44, -9.53, -2.29) mm, rotated rx -179.9 ry 0 rz -90 deg; joints [41.481, -70.962, 113.508, -126.752, 55.744, 144.029]
  MoveL 492 to (331.4, -9.52, -1.95) mm, rotated rx -179.9 ry 0 rz -90 deg; joints [41.49, -70.979, 113.531, -126.747, 55.753, 144.031]
  MoveL 493 to (331.35, -9.53, -1.6) mm, rotated rx -179.9 ry 0 rz -90 deg; joints [41.498, -70.996, 113.555, -126.743, 55.762, 144.033]
  MoveL 494 to (331.28, -9.52, -1.25) mm, rotated rx -179.9 ry 0 rz -90 deg; joints [41.506, -71.015, 113.58, -126.739, 55.77, 144.035]
  MoveL 495 to (331.14, -9.53, -0.76) mm, rotated rx -179.9 ry 0 rz -90 deg; joints [41.515, -71.042, 113.617, -126.735, 55.782, 144.04]
  MoveL 496 to (330.96, -9.53, -0.28) mm, rotated rx -179.9 ry 0 rz -90 deg; joints [41.523, -71.07, 113.656, -126.733, 55.793, 144.046]
  MoveL 497 to (330.73, -9.52, 0.21) mm, rotated rx -179.9 ry 0 rz -90 deg; joints [41.53, -71.1, 113.698, -126.733, 55.803, 144.053]
  MoveL 498 to (330.59, -9.52, 0.45) mm, rotated rx -179.9 ry 0 rz -90 deg; joints [41.532, -71.116, 113.72, -126.734, 55.809, 144.058]
  MoveL 499 to (330.44, -9.52, 0.69) mm, rotated rx -179.9 ry 0 rz -90 deg; joints [41.535, -71.133, 113.743, -126.735, 55.814, 144.063]
  MoveL 500 to (330.15, -9.53, 1.12) mm, rotated rx -179.9 ry 0 rz -90 deg; joints [41.537, -71.163, 113.784, -126.739, 55.822, 144.072]
  MoveL 501 to (329.98, -9.53, 1.33) mm, rotated rx -179.9 ry 0 rz -90 deg; joints [41.538, -71.179, 113.807, -126.741, 55.826, 144.078]
  MoveL 502 to (329.79, -9.52, 1.54) mm, rotated rx -179.9 ry 0 rz -90 deg; joints [41.538, -71.196, 113.829, -126.745, 55.83, 144.084]
  MoveL 503 to (329.52, -9.53, 1.82) mm, rotated rx -179.9 ry 0 rz -90 deg; joints [41.537, -71.218, 113.86, -126.75, 55.834, 144.092]
  MoveL 504 to (329.26, -9.53, 2.06) mm, rotated rx -179.9 ry 0 rz -90 deg; joints [41.535, -71.24, 113.889, -126.756, 55.838, 144.101]
  MoveL 505 to (328.99, -9.53, 2.28) mm, rotated rx -179.9 ry 0 rz -90 deg; joints [41.533, -71.259, 113.917, -126.762, 55.841, 144.11]
  MoveL 506 to (328.72, -9.53, 2.47) mm, rotated rx -179.9 ry 0 rz -90 deg; joints [41.53, -71.278, 113.943, -126.769, 55.844, 144.118]
  MoveL 507 to (328.46, -9.53, 2.65) mm, rotated rx -179.9 ry 0 rz -90 deg; joints [41.526, -71.297, 113.968, -126.776, 55.846, 144.127]
  MoveL 508 to (328.19, -9.52, 2.81) mm, rotated rx -179.9 ry 0 rz -90 deg; joints [41.522, -71.314, 113.992, -126.784, 55.847, 144.135]
  MoveL 509 to (327.92, -9.52, 2.95) mm, rotated rx -179.9 ry 0 rz -90 deg; joints [41.518, -71.33, 114.015, -126.792, 55.848, 144.144]
  MoveL 510 to (327.66, -9.52, 3.07) mm, rotated rx -179.9 ry 0 rz -90 deg; joints [41.513, -71.346, 114.037, -126.8, 55.849, 144.152]
  MoveL 511 to (327.31, -9.53, 3.21) mm, rotated rx -179.9 ry 0 rz -90 deg; joints [41.505, -71.366, 114.064, -126.811, 55.849, 144.164]
  MoveL 512 to (326.96, -9.52, 3.33) mm, rotated rx -179.9 ry 0 rz -90 deg; joints [41.498, -71.385, 114.09, -126.823, 55.849, 144.175]
  MoveL 513 to (326.61, -9.52, 3.42) mm, rotated rx -179.9 ry 0 rz -90 deg; joints [41.489, -71.402, 114.115, -126.835, 55.848, 144.186]
  MoveL 514 to (326.26, -9.53, 3.5) mm, rotated rx -179.9 ry 0 rz -90 deg; joints [41.48, -71.419, 114.138, -126.848, 55.847, 144.197]
  MoveL 515 to (325.91, -9.53, 3.55) mm, rotated rx -179.9 ry 0 rz -90 deg; joints [41.47, -71.435, 114.16, -126.86, 55.845, 144.208]
  MoveL 516 to (325.56, -9.53, 3.59) mm, rotated rx -179.9 ry 0 rz -90 deg; joints [41.46, -71.45, 114.181, -126.874, 55.842, 144.219]
  MoveL 517 to (324.87, -9.52, 3.61) mm, rotated rx -179.9 ry 0 rz -90 deg; joints [41.438, -71.478, 114.219, -126.901, 55.836, 144.242]
  MoveL 518 to (319.99, -9.52, 3.61) mm, rotated rx -179.9 ry 0 rz -90 deg; joints [41.279, -71.666, 114.482, -127.097, 55.787, 144.398]
  MoveL 519 to (319.81, -9.52, 3.73) mm, rotated rx -179.9 ry 0 rz -90 deg; joints [41.277, -71.679, 114.498, -127.101, 55.788, 144.403]
  MoveL 520 to (319.64, -9.52, 3.88) mm, rotated rx -179.9 ry 0 rz -90 deg; joints [41.275, -71.692, 114.517, -127.105, 55.791, 144.409]
  MoveL 521 to (319.29, -9.53, 4.15) mm, rotated rx -179.9 ry 0 rz -90 deg; joints [41.272, -71.717, 114.552, -127.114, 55.794, 144.42]
  MoveL 522 to (319.03, -9.52, 4.33) mm, rotated rx -179.9 ry 0 rz -90 deg; joints [41.268, -71.736, 114.577, -127.121, 55.796, 144.428]
  MoveL 523 to (318.71, -9.52, 4.52) mm, rotated rx -179.9 ry 0 rz -90 deg; joints [41.263, -71.756, 114.605, -127.13, 55.798, 144.438]
  MoveL 524 to (318.4, -9.52, 4.69) mm, rotated rx -179.9 ry 0 rz -90 deg; joints [41.258, -71.776, 114.632, -127.139, 55.799, 144.448]
  MoveL 525 to (318.08, -9.52, 4.84) mm, rotated rx -179.9 ry 0 rz -90 deg; joints [41.252, -71.794, 114.658, -127.149, 55.8, 144.458]
  MoveL 526 to (317.76, -9.53, 4.96) mm, rotated rx -179.9 ry 0 rz -90 deg; joints [41.245, -71.812, 114.682, -127.159, 55.8, 144.468]
  MoveL 527 to (317.45, -9.52, 5.07) mm, rotated rx -179.9 ry 0 rz -90 deg; joints [41.238, -71.829, 114.705, -127.17, 55.8, 144.478]
  MoveL 528 to (317.13, -9.52, 5.16) mm, rotated rx -179.9 ry 0 rz -90 deg; joints [41.23, -71.845, 114.727, -127.181, 55.799, 144.488]
  MoveL 529 to (316.82, -9.52, 5.23) mm, rotated rx -179.9 ry 0 rz -90 deg; joints [41.222, -71.861, 114.749, -127.192, 55.797, 144.498]
  MoveL 530 to (316.5, -9.53, 5.28) mm, rotated rx -179.9 ry 0 rz -90 deg; joints [41.213, -71.875, 114.769, -127.204, 55.796, 144.508]
  MoveL 531 to (316.15, -9.53, 5.32) mm, rotated rx -179.9 ry 0 rz -90 deg; joints [41.203, -71.89, 114.79, -127.217, 55.793, 144.519]
  MoveL 532 to (315.8, -9.52, 5.35) mm, rotated rx -179.9 ry 0 rz -90 deg; joints [41.192, -71.905, 114.81, -127.23, 55.79, 144.53]
  MoveL 533 to (315.11, -9.53, 5.35) mm, rotated rx -179.9 ry 0 rz -90 deg; joints [41.169, -71.932, 114.847, -127.258, 55.783, 144.553]
  MoveL 534 to (-302.56, -9.53, 5.35) mm, rotated rx -179.9 ry 0 rz -90 deg; joints [14.024, -90.069, 136.685, -160.755, 47.301, 167.125]
  MoveL 535 to (-303.26, -9.53, 5.35) mm, rotated rx -179.9 ry 0 rz -90 deg; joints [13.986, -90.08, 136.696, -160.805, 47.292, 167.159]
  MoveL 536 to (-303.6, -9.53, 5.33) mm, rotated rx -179.9 ry 0 rz -90 deg; joints [13.967, -90.085, 136.701, -160.831, 47.288, 167.176]
  MoveL 537 to (-303.95, -9.53, 5.29) mm, rotated rx -179.9 ry 0 rz -90 deg; joints [13.947, -90.088, 136.704, -160.857, 47.284, 167.193]
  MoveL 538 to (-304.3, -9.52, 5.23) mm, rotated rx -179.9 ry 0 rz -90 deg; joints [13.927, -90.089, 136.706, -160.883, 47.279, 167.211]
  MoveL 539 to (-304.65, -9.53, 5.15) mm, rotated rx -179.9 ry 0 rz -90 deg; joints [13.907, -90.09, 136.706, -160.91, 47.275, 167.229]
  MoveL 540 to (-305, -9.53, 5.05) mm, rotated rx -179.9 ry 0 rz -90 deg; joints [13.887, -90.089, 136.706, -160.937, 47.271, 167.247]
  MoveL 541 to (-305.35, -9.52, 4.92) mm, rotated rx -179.9 ry 0 rz -90 deg; joints [13.866, -90.086, 136.703, -160.965, 47.266, 167.265]
  MoveL 542 to (-305.64, -9.52, 4.8) mm, rotated rx -179.9 ry 0 rz -90 deg; joints [13.849, -90.083, 136.7, -160.988, 47.263, 167.281]
  MoveL 543 to (-305.93, -9.52, 4.67) mm, rotated rx -179.9 ry 0 rz -90 deg; joints [13.831, -90.078, 136.696, -161.012, 47.259, 167.297]
  MoveL 544 to (-306.22, -9.53, 4.51) mm, rotated rx -179.9 ry 0 rz -90 deg; joints [13.813, -90.073, 136.691, -161.036, 47.255, 167.313]
  MoveL 545 to (-306.51, -9.53, 4.33) mm, rotated rx -179.9 ry 0 rz -90 deg; joints [13.795, -90.065, 136.684, -161.06, 47.252, 167.329]
  MoveL 546 to (-306.92, -9.52, 4.05) mm, rotated rx -179.9 ry 0 rz -90 deg; joints [13.768, -90.053, 136.672, -161.095, 47.246, 167.353]
  MoveL 547 to (-307.32, -9.52, 3.71) mm, rotated rx -179.9 ry 0 rz -90 deg; joints [13.742, -90.037, 136.657, -161.13, 47.241, 167.377]
  MoveL 548 to (-307.53, -9.53, 3.61) mm, rotated rx -179.9 ry 0 rz -90 deg; joints [13.729, -90.034, 136.653, -161.147, 47.238, 167.388]
  MoveL 549 to (-308.14, -9.52, 3.61) mm, rotated rx -179.9 ry 0 rz -90 deg; joints [13.696, -90.043, 136.663, -161.191, 47.231, 167.417]
  MoveC 550 to (-309.11, -9.53, 4.07) mm, rotated rx -179.9 ry 0 rz -90 deg; joints [13.649, -90.089, 136.709, -161.254, 47.22, 167.459] to (-309.38, -9.53, 5.11) mm, rotated rx -179.9 ry 0 rz -90 deg; joints [13.648, -90.163, 136.781, -161.255, 47.219, 167.459]
  MoveL 551 to (-309.38, -9.52, 5.11) mm, rotated rx -179.9 ry 0 rz -90 deg; joints [13.648, -90.163, 136.781, -161.255, 47.219, 167.459]
  MoveL 552 to (-308.43, -9.52, 10.09) mm, rotated rx -179.9 ry 0 rz -90 deg; joints [13.767, -90.479, 137.088, -161.094, 47.236, 167.349]
  MoveL 553 to (-308.2, -8.25, 11.34) mm, rotated rx -179.9 ry 0 rz -90 deg; joints [13.797, -90.621, 137.117, -161.021, 47.136, 167.273]
  Set speed (200.0 mm/s)
  MoveL 554 to (-308.2, 25.52, 11.34) mm, rotated rx -179.9 ry 0 rz -90 deg; joints [13.782, -92.211, 135.82, -160.105, 44.41, 165.946]
  Print: /'90 deg cut'
  Call SetTool(1)
  Set speed (200.0 mm/s)
  MoveL 555 to (-315.82, 25.52, -1.73) mm, rotated rx -179.9 ry 0 rz -90 deg; joints [13.192, -91.448, 135.107, -160.941, 44.315, 166.546]
  MoveL 556 to (-315.82, 12.35, -1.73) mm, rotated rx -179.9 ry 0 rz -90 deg; joints [13.197, -90.85, 135.619, -161.295, 45.367, 167.05]
  Set speed (50.0 mm/s)
  MoveL 557 to (-315.82, 5.79, -1.73) mm, rotated rx -179.9 ry 0 rz -90 deg; joints [13.2, -90.544, 135.869, -161.465, 45.894, 167.296]
  MoveL 558 to (-314.58, 4.52, -1.45) mm, rotated rx -179.9 ry 0 rz -90 deg; joints [13.272, -90.484, 135.916, -161.4, 46.011, 167.277]
  Set speed (100.0 mm/s)
  MoveL 559 to (-310.96, 4.53, -0.65) mm, rotated rx -179.9 ry 0 rz -90 deg; joints [13.48, -90.481, 135.91, -161.118, 46.056, 167.084]
  MoveC 560 to (-309.89, 4.52, -0.9) mm, rotated rx -179.9 ry 0 rz -90 deg; joints [13.535, -90.447, 135.877, -161.044, 46.069, 167.033] to (-309.41, 4.53, -1.89) mm, rotated rx -179.9 ry 0 rz -90 deg; joints [13.547, -90.374, 135.806, -161.027, 46.073, 167.022]
  MoveL 561 to (-309.41, 4.53, -1.89) mm, rotated rx -179.9 ry 0 rz -90 deg; joints [13.547, -90.374, 135.806, -161.027, 46.073, 167.022]
  MoveL 562 to (-309.41, 4.53, -310.95) mm, rotated rx -179.9 ry 0 rz -90 deg; joints [10.396, -71.44, 113.629, -164.456, 42.303, 168.759]
  MoveL 563 to (-309.4, 4.52, -311.59) mm, rotated rx -179.9 ry 0 rz -90 deg; joints [10.391, -71.402, 113.578, -164.459, 42.289, 168.758]
  MoveL 564 to (-309.38, 4.52, -311.91) mm, rotated rx -179.9 ry 0 rz -90 deg; joints [10.39, -71.383, 113.552, -164.459, 42.282, 168.757]
  MoveL 565 to (-309.36, 4.52, -312.07) mm, rotated rx -179.9 ry 0 rz -90 deg; joints [10.389, -71.373, 113.539, -164.458, 42.278, 168.756]
  MoveC 566 to (-309.71, 4.52, -313.11) mm, rotated rx -179.9 ry 0 rz -90 deg; joints [10.366, -71.316, 113.461, -164.486, 42.254, 168.772] to (-310.74, 4.53, -313.49) mm, rotated rx -179.9 ry 0 rz -90 deg; joints [10.319, -71.305, 113.447, -164.553, 42.241, 168.821]
  MoveL 567 to (-310.74, 4.52, -313.49) mm, rotated rx -179.9 ry 0 rz -90 deg; joints [10.319, -71.305, 113.447, -164.553, 42.241, 168.821]
  MoveL 568 to (-314.43, 4.52, -313.12) mm, rotated rx -179.9 ry 0 rz -90 deg; joints [10.166, -71.365, 113.53, -164.784, 42.234, 168.994]
  MoveL 569 to (-315.69, 5.79, -313) mm, rotated rx -179.9 ry 0 rz -90 deg; joints [10.112, -71.431, 113.518, -164.839, 42.149, 169.02]
  Set speed (200.0 mm/s)
  MoveL 570 to (-315.69, 12.6, -313) mm, rotated rx -179.9 ry 0 rz -90 deg; joints [10.111, -71.673, 113.302, -164.708, 41.706, 168.842]
  MoveL 571 to (-316.7, 12.6, -1.92) mm, rotated rx -179.9 ry 0 rz -90 deg; joints [13.146, -90.862, 135.611, -161.358, 45.336, 167.089]
  MoveL 572 to (-316.7, 7, -1.92) mm, rotated rx -179.9 ry 0 rz -90 deg; joints [13.149, -90.602, 135.825, -161.503, 45.786, 167.299]
  Set speed (50.0 mm/s)
  MoveL 573 to (-316.7, 1.27, -1.92) mm, rotated rx -179.9 ry 0 rz -90 deg; joints [13.151, -90.331, 136.041, -161.648, 46.248, 167.51]
  MoveL 574 to (-315.46, 0, -1.65) mm, rotated rx -179.9 ry 0 rz -90 deg; joints [13.223, -90.27, 136.087, -161.584, 46.365, 167.491]
  Set speed (100.0 mm/s)
  MoveL 575 to (-310.96, 0, -0.65) mm, rotated rx -179.9 ry 0 rz -90 deg; joints [13.481, -90.266, 136.08, -161.235, 46.42, 167.254]
  MoveC 576 to (-309.89, 0, -0.9) mm, rotated rx -179.9 ry 0 rz -90 deg; joints [13.536, -90.233, 136.047, -161.161, 46.433, 167.204] to (-309.41, 0, -1.89) mm, rotated rx -179.9 ry 0 rz -90 deg; joints [13.549, -90.159, 135.975, -161.144, 46.437, 167.193]
  MoveL 577 to (-309.41, 0, -1.89) mm, rotated rx -179.9 ry 0 rz -90 deg; joints [13.549, -90.159, 135.975, -161.144, 46.437, 167.193]
  MoveL 578 to (-309.41, 0, -310.95) mm, rotated rx -179.9 ry 0 rz -90 deg; joints [10.397, -71.276, 113.77, -164.543, 42.597, 168.878]
  MoveL 579 to (-309.4, 0, -311.59) mm, rotated rx -179.9 ry 0 rz -90 deg; joints [10.392, -71.238, 113.719, -164.546, 42.583, 168.877]
  MoveL 580 to (-309.38, 0, -311.91) mm, rotated rx -179.9 ry 0 rz -90 deg; joints [10.391, -71.219, 113.693, -164.546, 42.576, 168.876]
  MoveL 581 to (-309.36, 0, -312.07) mm, rotated rx -179.9 ry 0 rz -90 deg; joints [10.391, -71.21, 113.68, -164.546, 42.572, 168.875]
  MoveC 582 to (-309.71, 0, -313.11) mm, rotated rx -179.9 ry 0 rz -90 deg; joints [10.367, -71.153, 113.603, -164.573, 42.548, 168.892] to (-310.74, 0, -313.49) mm, rotated rx -179.9 ry 0 rz -90 deg; joints [10.321, -71.142, 113.588, -164.64, 42.535, 168.939]
  MoveL 583 to (-310.74, 0, -313.49) mm, rotated rx -179.9 ry 0 rz -90 deg; joints [10.321, -71.142, 113.588, -164.64, 42.535, 168.939]
  MoveL 584 to (-315.33, 0, -313.03) mm, rotated rx -179.9 ry 0 rz -90 deg; joints [10.129, -71.216, 113.692, -164.926, 42.527, 169.152]
  MoveL 585 to (-316.6, 1.27, -312.91) mm, rotated rx -179.9 ry 0 rz -90 deg; joints [10.076, -71.282, 113.68, -164.981, 42.442, 169.179]
  Set speed (200.0 mm/s)
  MoveL 586 to (-316.6, 16.53, -312.91) mm, rotated rx -179.9 ry 0 rz -90 deg; joints [10.072, -71.826, 113.196, -164.688, 41.448, 168.781]
  MoveL 587 to (328.21, 16.53, -313) mm, rotated rx -179.9 ry 0 rz -90 deg; joints [33.853, -57.061, 90.925, -128.889, 45.686, 139.941]
  MoveL 588 to (328.21, 12.35, -313) mm, rotated rx -179.9 ry 0 rz -90 deg; joints [33.855, -56.948, 91.058, -129.073, 45.842, 140.206]
  Set speed (50.0 mm/s)
  MoveL 589 to (328.21, 5.8, -313) mm, rotated rx -179.9 ry 0 rz -90 deg; joints [33.858, -56.769, 91.264, -129.358, 46.087, 140.619]
  MoveL 590 to (326.95, 4.53, -313.12) mm, rotated rx -179.9 ry 0 rz -90 deg; joints [33.818, -56.771, 91.364, -129.474, 46.124, 140.753]
  Set speed (100.0 mm/s)
  MoveL 591 to (323.26, 4.52, -313.49) mm, rotated rx -179.9 ry 0 rz -90 deg; joints [33.699, -56.879, 91.54, -129.652, 46.092, 140.912]
  MoveC 592 to (322.23, 4.53, -313.11) mm, rotated rx -179.9 ry 0 rz -90 deg; joints [33.675, -56.934, 91.628, -129.702, 46.098, 140.965] to (321.87, 4.53, -312.07) mm, rotated rx -179.9 ry 0 rz -90 deg; joints [33.685, -57, 91.734, -129.72, 46.13, 141]
  MoveL 593 to (321.87, 4.52, -312.07) mm, rotated rx -179.9 ry 0 rz -90 deg; joints [33.685, -57, 91.734, -129.72, 46.13, 141]
  MoveL 594 to (321.89, 4.52, -311.91) mm, rotated rx -179.9 ry 0 rz -90 deg; joints [33.689, -57.008, 91.746, -129.719, 46.135, 141.002]
  MoveL 595 to (321.92, 4.52, -311.59) mm, rotated rx -179.9 ry 0 rz -90 deg; joints [33.696, -57.024, 91.771, -129.718, 46.145, 141.006]
  MoveL 596 to (321.93, 4.52, -310.95) mm, rotated rx -179.9 ry 0 rz -90 deg; joints [33.71, -57.057, 91.823, -129.718, 46.166, 141.017]
  MoveL 597 to (321.93, 4.53, -1.89) mm, rotated rx -179.9 ry 0 rz -90 deg; joints [41.176, -71.858, 113.61, -126.611, 55.088, 143.419]
  MoveC 598 to (322.4, 4.52, -0.9) mm, rotated rx -179.9 ry 0 rz -90 deg; joints [41.22, -71.884, 113.644, -126.573, 55.119, 143.404] to (323.47, 4.52, -0.65) mm, rotated rx -179.9 ry 0 rz -90 deg; joints [41.262, -71.854, 113.602, -126.525, 55.137, 143.369]
  MoveL 599 to (323.47, 4.53, -0.65) mm, rotated rx -179.9 ry 0 rz -90 deg; joints [41.262, -71.854, 113.602, -126.525, 55.137, 143.369]
  MoveL 600 to (327.09, 4.52, -1.45) mm, rotated rx -179.9 ry 0 rz -90 deg; joints [41.356, -71.677, 113.359, -126.396, 55.155, 143.253]
  MoveL 601 to (328.33, 5.79, -1.73) mm, rotated rx -179.9 ry 0 rz -90 deg; joints [41.388, -71.662, 113.235, -126.304, 55.109, 143.13]
  Set speed (200.0 mm/s)
  MoveL 602 to (328.33, 12.35, -1.73) mm, rotated rx -179.9 ry 0 rz -90 deg; joints [41.384, -71.894, 113.026, -126.058, 54.846, 142.697]
  MoveL 603 to (329.11, 12.35, -312.91) mm, rotated rx -179.9 ry 0 rz -90 deg; joints [33.884, -56.922, 91.015, -129.029, 45.85, 140.167]
  MoveL 604 to (329.11, 7, -312.91) mm, rotated rx -179.9 ry 0 rz -90 deg; joints [33.886, -56.776, 91.183, -129.262, 46.05, 140.504]
  Set speed (50.0 mm/s)
  MoveL 605 to (329.11, 1.27, -312.91) mm, rotated rx -179.9 ry 0 rz -90 deg; joints [33.889, -56.617, 91.361, -129.509, 46.265, 140.863]
  MoveL 606 to (327.85, 0, -313.03) mm, rotated rx -179.9 ry 0 rz -90 deg; joints [33.849, -56.619, 91.46, -129.624, 46.302, 140.996]
  Set speed (100.0 mm/s)
  MoveL 607 to (323.26, 0, -313.49) mm, rotated rx -179.9 ry 0 rz -90 deg; joints [33.701, -56.753, 91.679, -129.845, 46.262, 141.193]
  MoveC 608 to (322.23, 0, -313.11) mm, rotated rx -179.9 ry 0 rz -90 deg; joints [33.677, -56.808, 91.767, -129.895, 46.269, 141.246] to (321.87, 0, -312.07) mm, rotated rx -179.9 ry 0 rz -90 deg; joints [33.687, -56.874, 91.873, -129.913, 46.301, 141.281]
  MoveL 609 to (321.87, 0, -312.07) mm, rotated rx -179.9 ry 0 rz -90 deg; joints [33.687, -56.874, 91.873, -129.913, 46.301, 141.281]
  MoveL 610 to (321.89, 0, -311.91) mm, rotated rx -179.9 ry 0 rz -90 deg; joints [33.691, -56.882, 91.885, -129.912, 46.306, 141.283]
  MoveL 611 to (321.92, 0, -311.59) mm, rotated rx -179.9 ry 0 rz -90 deg; joints [33.698, -56.897, 91.91, -129.911, 46.317, 141.287]
  MoveL 612 to (321.93, 0, -310.95) mm, rotated rx -179.9 ry 0 rz -90 deg; joints [33.712, -56.93, 91.962, -129.911, 46.338, 141.298]
  MoveL 613 to (321.93, 0, -1.89) mm, rotated rx -179.9 ry 0 rz -90 deg; joints [41.179, -71.695, 113.752, -126.778, 55.272, 143.716]
  MoveC 614 to (322.4, 0, -0.9) mm, rotated rx -179.9 ry 0 rz -90 deg; joints [41.223, -71.721, 113.786, -126.74, 55.303, 143.7] to (323.47, 0, -0.65) mm, rotated rx -179.9 ry 0 rz -90 deg; joints [41.265, -71.691, 113.744, -126.692, 55.321, 143.666]
  MoveL 615 to (323.47, 0, -0.65) mm, rotated rx -179.9 ry 0 rz -90 deg; joints [41.265, -71.691, 113.744, -126.692, 55.321, 143.666]
  MoveL 616 to (327.98, 0, -1.65) mm, rotated rx -179.9 ry 0 rz -90 deg; joints [41.382, -71.471, 113.441, -126.532, 55.341, 143.521]
  MoveL 617 to (329.22, 1.27, -1.92) mm, rotated rx -179.9 ry 0 rz -90 deg; joints [41.414, -71.457, 113.318, -126.44, 55.295, 143.398]
  Set speed (200.0 mm/s)
  MoveL 618 to (329.22, 25.53, -1.92) mm, rotated rx -179.9 ry 0 rz -90 deg; joints [41.399, -72.307, 112.536, -125.523, 54.328, 141.79]
  Print: /'diagnonal cut'
  Call SetTool(1)
  Set speed (200.0 mm/s)
  MoveL 619 to (-335.6, -11.85, 4.35) mm, rotated rx -179.15 ry 0 rz -30.08 deg; joints [-4.556, -80.871, 143.724, -185.5, 62.768, 242.639]
  MoveL 620 to (-332.9, -13.41, 4.35) mm, rotated rx -179.15 ry 0 rz -30.08 deg; joints [-4.4, -80.769, 143.771, -185.317, 62.91, 242.544]
  Set speed (50.0 mm/s)
  MoveL 621 to (-326.98, -16.84, 4.35) mm, rotated rx -179.15 ry 0 rz -30.08 deg; joints [-4.057, -80.541, 143.871, -184.918, 63.223, 242.338]
  MoveL 622 to (-325.36, -16.57, 3.64) mm, rotated rx -179.15 ry 0 rz -30.08 deg; joints [-3.96, -80.527, 143.822, -184.811, 63.185, 242.293]
  Set speed (100.0 mm/s)
  MoveL 623 to (-324.39, -14.89, 2.31) mm, rotated rx -179.15 ry 0 rz -30.08 deg; joints [-3.899, -80.579, 143.698, -184.75, 63.007, 242.279]
  MoveC 624 to (-324.11, -14.42, 1.33) mm, rotated rx -179.15 ry 0 rz -30.08 deg; joints [-3.879, -80.559, 143.62, -184.731, 62.949, 242.274] to (-324.33, -14.8, 0.3) mm, rotated rx -179.15 ry 0 rz -30.08 deg; joints [-3.888, -80.472, 143.554, -184.74, 62.97, 242.277]
  MoveL 625 to (-324.33, -14.8, 0.3) mm, rotated rx -179.15 ry 0 rz -30.08 deg; joints [-3.888, -80.472, 143.554, -184.74, 62.97, 242.277]
  MoveL 626 to (-324.51, -15.11, -0.05) mm, rotated rx -179.15 ry 0 rz -30.08 deg; joints [-3.897, -80.428, 143.535, -184.749, 62.995, 242.279]
  MoveL 627 to (-324.67, -15.38, -0.39) mm, rotated rx -179.15 ry 0 rz -30.08 deg; joints [-3.905, -80.388, 143.515, -184.757, 63.015, 242.281]
  MoveL 628 to (-324.81, -15.61, -0.73) mm, rotated rx -179.15 ry 0 rz -30.08 deg; joints [-3.911, -80.351, 143.495, -184.763, 63.032, 242.283]
  MoveL 629 to (-324.92, -15.82, -1.07) mm, rotated rx -179.15 ry 0 rz -30.08 deg; joints [-3.917, -80.316, 143.474, -184.769, 63.047, 242.284]
  MoveL 630 to (-325.03, -15.99, -1.42) mm, rotated rx -179.15 ry 0 rz -30.08 deg; joints [-3.921, -80.283, 143.453, -184.773, 63.058, 242.285]
  MoveL 631 to (-325.11, -16.15, -1.76) mm, rotated rx -179.15 ry 0 rz -30.08 deg; joints [-3.925, -80.253, 143.431, -184.777, 63.067, 242.286]
  MoveL 632 to (-325.19, -16.28, -2.1) mm, rotated rx -179.15 ry 0 rz -30.08 deg; joints [-3.928, -80.223, 143.409, -184.78, 63.075, 242.287]
  MoveL 633 to (-325.25, -16.39, -2.45) mm, rotated rx -179.15 ry 0 rz -30.08 deg; joints [-3.93, -80.195, 143.386, -184.783, 63.08, 242.288]
  MoveL 634 to (-325.31, -16.48, -2.8) mm, rotated rx -179.15 ry 0 rz -30.08 deg; joints [-3.932, -80.169, 143.363, -184.784, 63.084, 242.288]
  MoveL 635 to (-325.35, -16.55, -3.14) mm, rotated rx -179.15 ry 0 rz -30.08 deg; joints [-3.933, -80.143, 143.34, -184.786, 63.086, 242.289]
  MoveL 636 to (-325.38, -16.61, -3.49) mm, rotated rx -179.15 ry 0 rz -30.08 deg; joints [-3.934, -80.119, 143.316, -184.786, 63.086, 242.289]
  MoveL 637 to (-325.41, -16.65, -3.84) mm, rotated rx -179.15 ry 0 rz -30.08 deg; joints [-3.934, -80.096, 143.292, -184.786, 63.084, 242.289]
  MoveL 638 to (-325.42, -16.67, -4.19) mm, rotated rx -179.15 ry 0 rz -30.08 deg; joints [-3.933, -80.075, 143.267, -184.786, 63.081, 242.289]
  MoveL 639 to (-325.42, -16.68, -4.54) mm, rotated rx -179.15 ry 0 rz -30.08 deg; joints [-3.932, -80.055, 143.242, -184.785, 63.077, 242.289]
  MoveL 640 to (-325.42, -16.68, -311.19) mm, rotated rx -179.15 ry 0 rz -30.08 deg; joints [-3.029, -63.989, 119.926, -184.065, 55.813, 242.408]
  MoveL 641 to (-325.42, -16.67, -311.54) mm, rotated rx -179.15 ry 0 rz -30.08 deg; joints [-3.028, -63.971, 119.898, -184.064, 55.802, 242.409]
  MoveL 642 to (-325.41, -16.65, -311.88) mm, rotated rx -179.15 ry 0 rz -30.08 deg; joints [-3.026, -63.955, 119.869, -184.063, 55.79, 242.409]
  MoveL 643 to (-325.38, -16.61, -312.23) mm, rotated rx -179.15 ry 0 rz -30.08 deg; joints [-3.025, -63.939, 119.84, -184.062, 55.776, 242.409]
  MoveL 644 to (-325.35, -16.55, -312.58) mm, rotated rx -179.15 ry 0 rz -30.08 deg; joints [-3.022, -63.924, 119.81, -184.06, 55.761, 242.408]
  MoveL 645 to (-325.31, -16.48, -312.93) mm, rotated rx -179.15 ry 0 rz -30.08 deg; joints [-3.02, -63.911, 119.781, -184.057, 55.746, 242.408]
  MoveL 646 to (-325.25, -16.39, -313.28) mm, rotated rx -179.15 ry 0 rz -30.08 deg; joints [-3.017, -63.898, 119.751, -184.054, 55.729, 242.407]
  MoveL 647 to (-325.19, -16.27, -313.63) mm, rotated rx -179.15 ry 0 rz -30.08 deg; joints [-3.013, -63.886, 119.721, -184.051, 55.71, 242.406]
  MoveL 648 to (-325.11, -16.14, -313.98) mm, rotated rx -179.15 ry 0 rz -30.08 deg; joints [-3.009, -63.875, 119.691, -184.047, 55.691, 242.405]
  MoveL 649 to (-325.02, -15.98, -314.33) mm, rotated rx -179.15 ry 0 rz -30.08 deg; joints [-3.004, -63.866, 119.66, -184.042, 55.669, 242.404]
  MoveL 650 to (-324.91, -15.8, -314.68) mm, rotated rx -179.15 ry 0 rz -30.08 deg; joints [-2.999, -63.857, 119.629, -184.036, 55.647, 242.402]
  MoveL 651 to (-324.79, -15.59, -315.03) mm, rotated rx -179.15 ry 0 rz -30.08 deg; joints [-2.993, -63.851, 119.598, -184.03, 55.622, 242.4]
  MoveL 652 to (-324.65, -15.35, -315.38) mm, rotated rx -179.15 ry 0 rz -30.08 deg; joints [-2.986, -63.846, 119.566, -184.023, 55.595, 242.398]
  MoveL 653 to (-324.5, -15.09, -315.7) mm, rotated rx -179.15 ry 0 rz -30.08 deg; joints [-2.978, -63.843, 119.536, -184.016, 55.568, 242.395]
  MoveL 654 to (-324.33, -14.8, -316.02) mm, rotated rx -179.15 ry 0 rz -30.08 deg; joints [-2.97, -63.842, 119.506, -184.007, 55.538, 242.392]
  MoveL 655 to (-324.16, -14.49, -316.3) mm, rotated rx -179.15 ry 0 rz -30.08 deg; joints [-2.962, -63.843, 119.479, -183.999, 55.51, 242.389]
  MoveL 656 to (-323.98, -14.19, -316.55) mm, rotated rx -179.15 ry 0 rz -30.08 deg; joints [-2.954, -63.846, 119.455, -183.99, 55.482, 242.385]
  MoveL 657 to (-323.81, -13.89, -316.76) mm, rotated rx -179.15 ry 0 rz -30.08 deg; joints [-2.946, -63.851, 119.433, -183.982, 55.456, 242.382]
  MoveL 658 to (-323.63, -13.59, -316.94) mm, rotated rx -179.15 ry 0 rz -30.08 deg; joints [-2.938, -63.857, 119.414, -183.973, 55.43, 242.379]
  MoveL 659 to (-323.46, -13.29, -317.1) mm, rotated rx -179.15 ry 0 rz -30.08 deg; joints [-2.93, -63.865, 119.397, -183.965, 55.405, 242.375]
  MoveL 660 to (-323.28, -12.99, -317.23) mm, rotated rx -179.15 ry 0 rz -30.08 deg; joints [-2.922, -63.874, 119.382, -183.956, 55.381, 242.372]
  MoveL 661 to (-323.11, -12.68, -317.34) mm, rotated rx -179.15 ry 0 rz -30.08 deg; joints [-2.914, -63.884, 119.369, -183.948, 55.358, 242.368]
  MoveL 662 to (-322.93, -12.38, -317.43) mm, rotated rx -179.15 ry 0 rz -30.08 deg; joints [-2.906, -63.895, 119.358, -183.939, 55.335, 242.365]
  MoveL 663 to (-322.76, -12.08, -317.5) mm, rotated rx -179.15 ry 0 rz -30.08 deg; joints [-2.899, -63.907, 119.348, -183.931, 55.313, 242.361]
  MoveL 664 to (-322.58, -11.78, -317.55) mm, rotated rx -179.15 ry 0 rz -30.08 deg; joints [-2.891, -63.92, 119.34, -183.923, 55.292, 242.358]
  MoveL 665 to (-322.41, -11.48, -317.58) mm, rotated rx -179.15 ry 0 rz -30.08 deg; joints [-2.883, -63.934, 119.334, -183.914, 55.271, 242.354]
  MoveL 666 to (-322.23, -11.17, -317.59) mm, rotated rx -179.15 ry 0 rz -30.08 deg; joints [-2.876, -63.949, 119.329, -183.906, 55.251, 242.351]
  MoveL 667 to (-315.94, -0.31, -317.59) mm, rotated rx -179.15 ry 0 rz -30.08 deg; joints [-2.602, -64.504, 119.173, -183.604, 54.531, 242.216]
  MoveL 668 to (-315.59, 0.29, -317.58) mm, rotated rx -179.15 ry 0 rz -30.08 deg; joints [-2.586, -64.535, 119.165, -183.587, 54.491, 242.208]
  MoveL 669 to (-315.42, 0.6, -317.55) mm, rotated rx -179.15 ry 0 rz -30.08 deg; joints [-2.579, -64.552, 119.163, -183.579, 54.472, 242.204]
  MoveL 670 to (-315.24, 0.9, -317.5) mm, rotated rx -179.15 ry 0 rz -30.08 deg; joints [-2.571, -64.57, 119.162, -183.57, 54.454, 242.201]
  MoveL 671 to (-315.07, 1.2, -317.43) mm, rotated rx -179.15 ry 0 rz -30.08 deg; joints [-2.564, -64.589, 119.163, -183.562, 54.436, 242.197]
  MoveL 672 to (-314.89, 1.5, -317.34) mm, rotated rx -179.15 ry 0 rz -30.08 deg; joints [-2.556, -64.608, 119.166, -183.553, 54.418, 242.193]
  MoveL 673 to (-314.72, 1.8, -317.23) mm, rotated rx -179.15 ry 0 rz -30.08 deg; joints [-2.549, -64.629, 119.17, -183.545, 54.401, 242.189]
  MoveL 674 to (-314.54, 2.1, -317.1) mm, rotated rx -179.15 ry 0 rz -30.08 deg; joints [-2.542, -64.651, 119.176, -183.537, 54.385, 242.185]
  MoveL 675 to (-314.39, 2.36, -316.97) mm, rotated rx -179.15 ry 0 rz -30.08 deg; joints [-2.535, -64.671, 119.183, -183.53, 54.372, 242.181]
  MoveL 676 to (-314.24, 2.62, -316.82) mm, rotated rx -179.15 ry 0 rz -30.08 deg; joints [-2.529, -64.692, 119.192, -183.523, 54.36, 242.178]
  MoveL 677 to (-314.09, 2.88, -316.65) mm, rotated rx -179.15 ry 0 rz -30.08 deg; joints [-2.523, -64.714, 119.202, -183.515, 54.348, 242.174]
  MoveL 678 to (-313.95, 3.13, -316.45) mm, rotated rx -179.15 ry 0 rz -30.08 deg; joints [-2.517, -64.737, 119.214, -183.508, 54.336, 242.17]
  MoveL 679 to (-313.8, 3.39, -316.23) mm, rotated rx -179.15 ry 0 rz -30.08 deg; joints [-2.511, -64.761, 119.228, -183.501, 54.326, 242.167]
  MoveL 680 to (-313.65, 3.65, -315.98) mm, rotated rx -179.15 ry 0 rz -30.08 deg; joints [-2.505, -64.787, 119.244, -183.494, 54.316, 242.163]
  MoveL 681 to (-313.49, 3.92, -315.68) mm, rotated rx -179.15 ry 0 rz -30.08 deg; joints [-2.498, -64.817, 119.265, -183.487, 54.307, 242.159]
  MoveL 682 to (-313.35, 4.16, -315.38) mm, rotated rx -179.15 ry 0 rz -30.08 deg; joints [-2.493, -64.845, 119.286, -183.48, 54.3, 242.156]
  MoveL 683 to (-313.24, 4.35, -315.11) mm, rotated rx -179.15 ry 0 rz -30.08 deg; joints [-2.489, -64.868, 119.305, -183.475, 54.295, 242.153]
  MoveL 684 to (-313.14, 4.52, -314.85) mm, rotated rx -179.15 ry 0 rz -30.08 deg; joints [-2.485, -64.89, 119.324, -183.471, 54.292, 242.151]
  MoveL 685 to (-313.05, 4.68, -314.57) mm, rotated rx -179.15 ry 0 rz -30.08 deg; joints [-2.481, -64.913, 119.344, -183.467, 54.29, 242.149]
  MoveL 686 to (-312.97, 4.82, -314.28) mm, rotated rx -179.15 ry 0 rz -30.08 deg; joints [-2.478, -64.934, 119.365, -183.463, 54.289, 242.146]
  MoveL 687 to (-312.9, 4.95, -314) mm, rotated rx -179.15 ry 0 rz -30.08 deg; joints [-2.476, -64.955, 119.386, -183.46, 54.289, 242.144]
  MoveL 688 to (-312.83, 5.06, -313.72) mm, rotated rx -179.15 ry 0 rz -30.08 deg; joints [-2.473, -64.976, 119.408, -183.457, 54.29, 242.143]
  MoveL 689 to (-312.73, 5.24, -313.15) mm, rotated rx -179.15 ry 0 rz -30.08 deg; joints [-2.47, -65.014, 119.451, -183.452, 54.295, 242.14]
